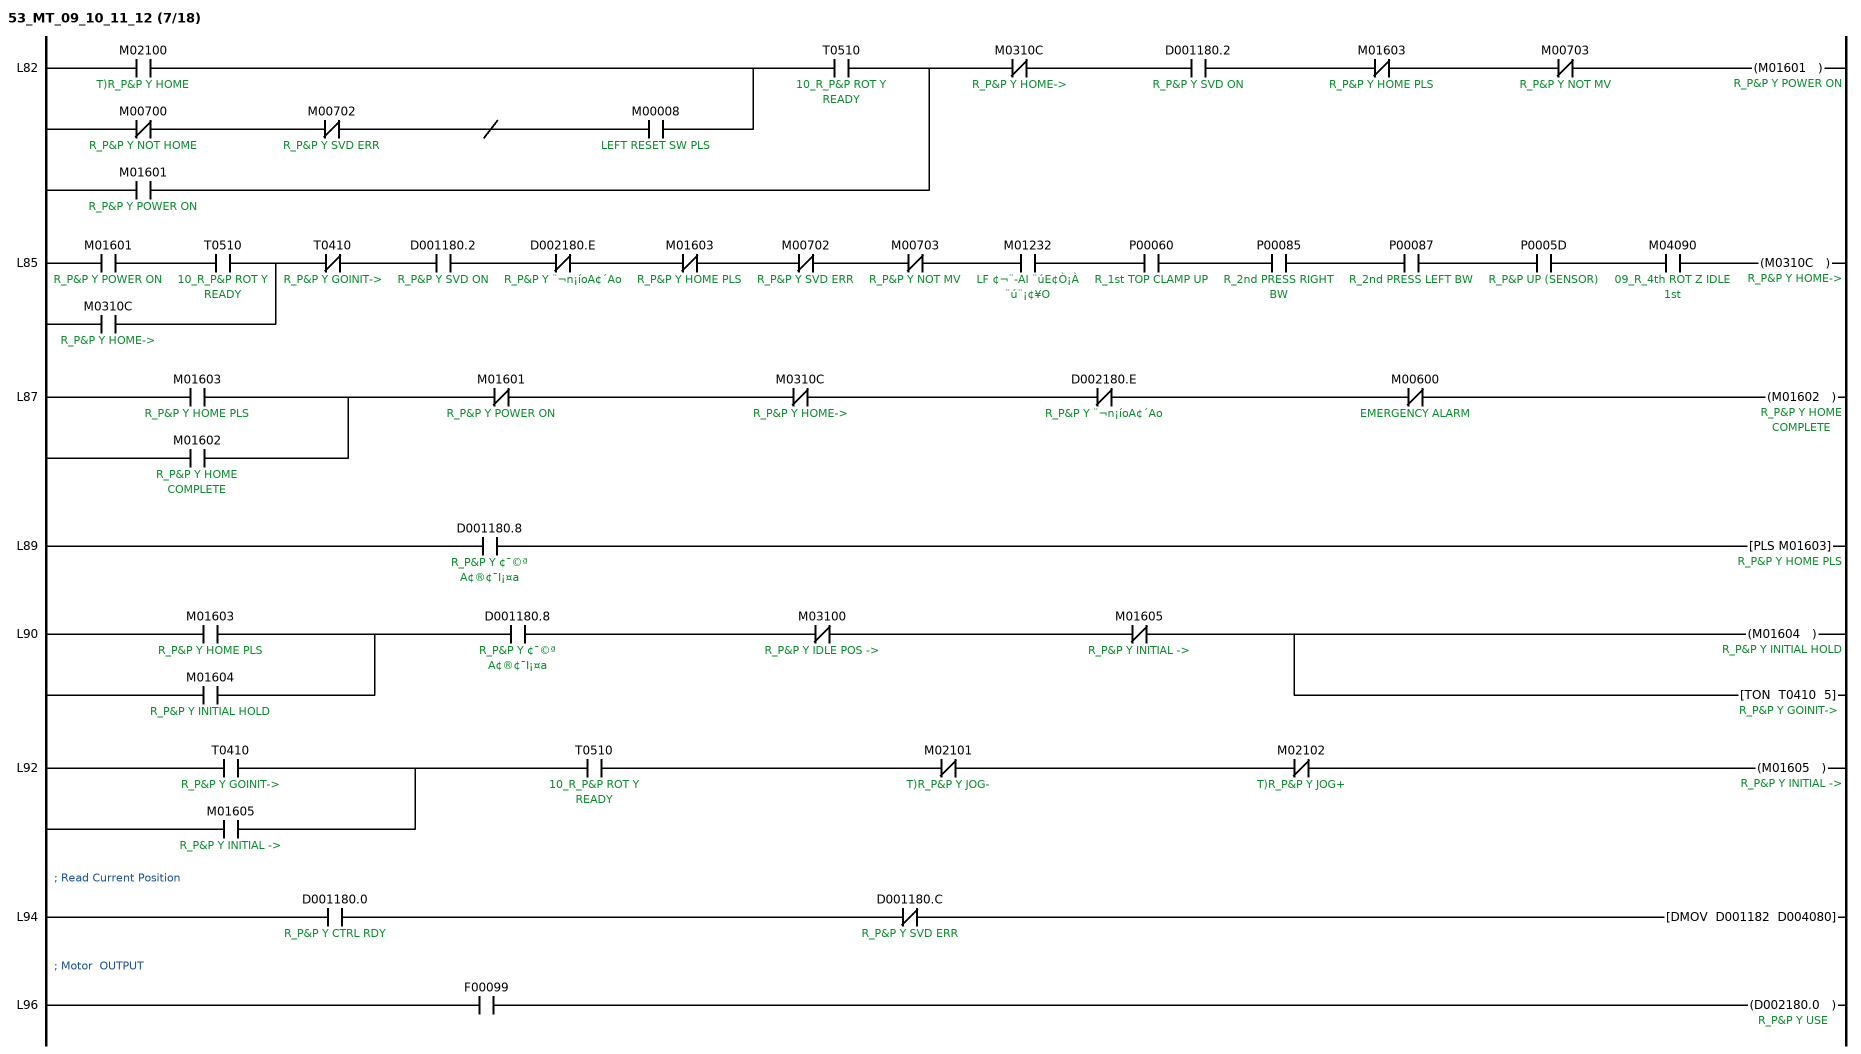
[picture p288: 53_MT_09_10_11_12 rungs L82-L96]
; L82
LOAD      M02100	// T)R_P&P Y HOME
LOAD NOT  M00700	// R_P&P Y NOT HOME
AND NOT   M00702	// R_P&P Y SVD ERR
NOT
AND       M00008	// LEFT RESET SW PLS
OR LOAD
AND       T0510	// 10_R_P&P ROT Y READY
OR        M01601	// R_P&P Y POWER ON
AND NOT   M0310C	// R_P&P Y HOME->
AND       D001180.2	// R_P&P Y SVD ON
AND NOT   M01603	// R_P&P Y HOME PLS
AND NOT   M00703	// R_P&P Y NOT MV
OUT       M01601	// R_P&P Y POWER ON
; L85
LOAD      M01601	// R_P&P Y POWER ON
AND       T0510	// 10_R_P&P ROT Y READY
OR        M0310C	// R_P&P Y HOME->
AND NOT   T0410	// R_P&P Y GOINIT->
AND       D001180.2	// R_P&P Y SVD ON
AND NOT   D002180.E	// R_P&P Y ¨¬n¡íoA¢´Ao
AND NOT   M01603	// R_P&P Y HOME PLS
AND NOT   M00702	// R_P&P Y SVD ERR
AND NOT   M00703	// R_P&P Y NOT MV
AND       M01232	// LF ¢¬¨­AI ¨úE¢Ò¡À ¨ú¨¡¢¥O
AND       P00060	// R_1st TOP CLAMP UP
AND       P00085	// R_2nd PRESS RIGHT BW
AND       P00087	// R_2nd PRESS LEFT BW
AND       P0005D	// R_P&P UP (SENSOR)
AND       M04090	// 09_R_4th ROT Z IDLE 1st
OUT       M0310C	// R_P&P Y HOME->
; L87
LOAD      M01603	// R_P&P Y HOME PLS
OR        M01602	// R_P&P Y HOME COMPLETE
AND NOT   M01601	// R_P&P Y POWER ON
AND NOT   M0310C	// R_P&P Y HOME->
AND NOT   D002180.E	// R_P&P Y ¨¬n¡íoA¢´Ao
AND NOT   M00600	// EMERGENCY ALARM
OUT       M01602	// R_P&P Y HOME COMPLETE
; L89
LOAD      D001180.8	// R_P&P Y ¢¯©ªA¢®¢¯I¡¤a
OUTP      M01603	// R_P&P Y HOME PLS
; L90
LOAD      M01603	// R_P&P Y HOME PLS
OR        M01604	// R_P&P Y INITIAL HOLD
AND       D001180.8	// R_P&P Y ¢¯©ªA¢®¢¯I¡¤a
AND NOT   M03100	// R_P&P Y IDLE POS ->
AND NOT   M01605	// R_P&P Y INITIAL ->
OUT       M01604	// R_P&P Y INITIAL HOLD
TON       T0410 5	// R_P&P Y GOINIT->
; L92
LOAD      T0410	// R_P&P Y GOINIT->
OR        M01605	// R_P&P Y INITIAL ->
AND       T0510	// 10_R_P&P ROT Y READY
AND NOT   M02101	// T)R_P&P Y JOG-
AND NOT   M02102	// T)R_P&P Y JOG+
OUT       M01605	// R_P&P Y INITIAL ->
; L94
LOAD      D001180.0	// R_P&P Y CTRL RDY
AND NOT   D001180.C	// R_P&P Y SVD ERR
DMOV      D001182 D004080
// output comment: Read Current Position
//  Motor  OUTPUT
; L96
LOAD      F00099
OUT       D002180.0	// R_P&P Y USE

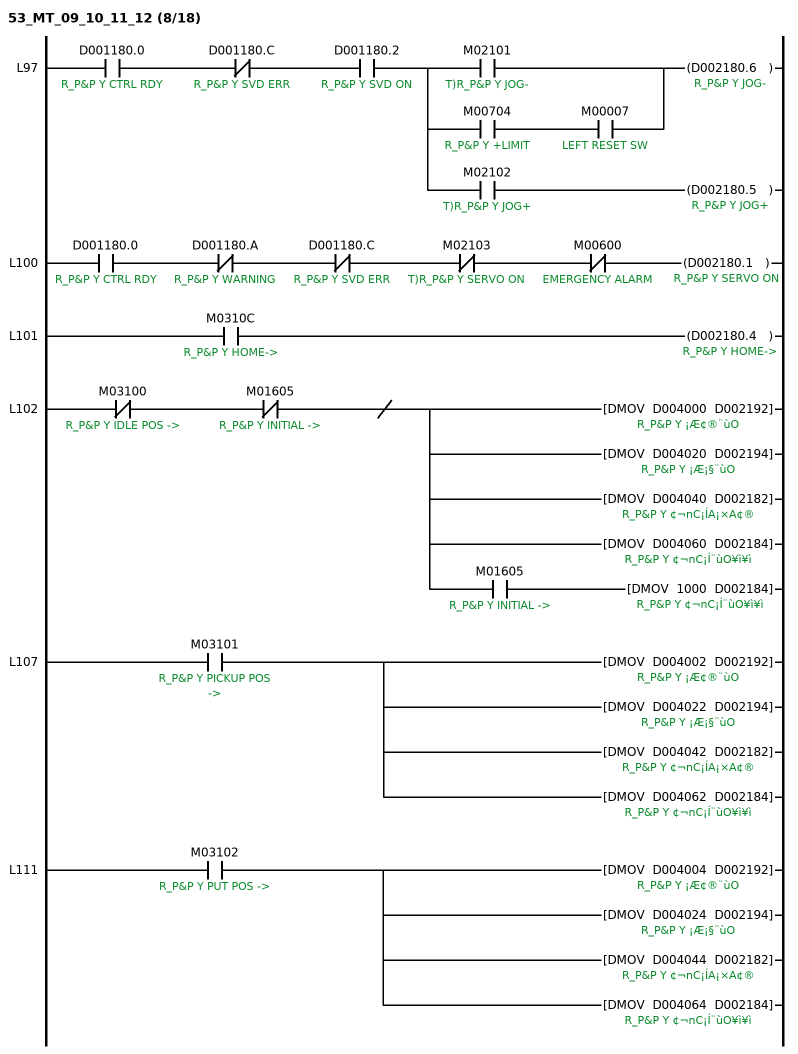
; L97
LOAD      D001180.0	// R_P&P Y CTRL RDY
AND NOT   D001180.C	// R_P&P Y SVD ERR
AND       D001180.2	// R_P&P Y SVD ON
MPUSH
LOAD      M02101	// T)R_P&P Y JOG-
LOAD      M00704	// R_P&P Y +LIMIT
AND       M00007	// LEFT RESET SW
OR LOAD
AND LOAD
OUT       D002180.6	// R_P&P Y JOG-
MPOP
AND       M02102	// T)R_P&P Y JOG+
OUT       D002180.5	// R_P&P Y JOG+
; L100
LOAD      D001180.0	// R_P&P Y CTRL RDY
AND NOT   D001180.A	// R_P&P Y WARNING
AND NOT   D001180.C	// R_P&P Y SVD ERR
AND NOT   M02103	// T)R_P&P Y SERVO ON
AND NOT   M00600	// EMERGENCY ALARM
OUT       D002180.1	// R_P&P Y SERVO ON
; L101
LOAD      M0310C	// R_P&P Y HOME->
OUT       D002180.4	// R_P&P Y HOME->
; L102
LOAD NOT  M03100	// R_P&P Y IDLE POS ->
AND NOT   M01605	// R_P&P Y INITIAL ->
NOT
DMOV      D004000 D002192	// R_P&P Y ¡Æ¢®¨ùO
DMOV      D004020 D002194	// R_P&P Y ¡Æ¡§¨ùO
DMOV      D004040 D002182	// R_P&P Y ¢¬nC¡ÍA¡×A¢®
DMOV      D004060 D002184	// R_P&P Y ¢¬nC¡Í¨ùO¥ì¥ì
AND       M01605	// R_P&P Y INITIAL ->
DMOV      1000 D002184	// R_P&P Y ¢¬nC¡Í¨ùO¥ì¥ì
; L107
LOAD      M03101	// R_P&P Y PICKUP POS ->
DMOV      D004002 D002192	// R_P&P Y ¡Æ¢®¨ùO
DMOV      D004022 D002194	// R_P&P Y ¡Æ¡§¨ùO
DMOV      D004042 D002182	// R_P&P Y ¢¬nC¡ÍA¡×A¢®
DMOV      D004062 D002184	// R_P&P Y ¢¬nC¡Í¨ùO¥ì¥ì
; L111
LOAD      M03102	// R_P&P Y PUT POS ->
DMOV      D004004 D002192	// R_P&P Y ¡Æ¢®¨ùO
DMOV      D004024 D002194	// R_P&P Y ¡Æ¡§¨ùO
DMOV      D004044 D002182	// R_P&P Y ¢¬nC¡ÍA¡×A¢®
DMOV      D004064 D002184	// R_P&P Y ¢¬nC¡Í¨ùO¥ì¥ì

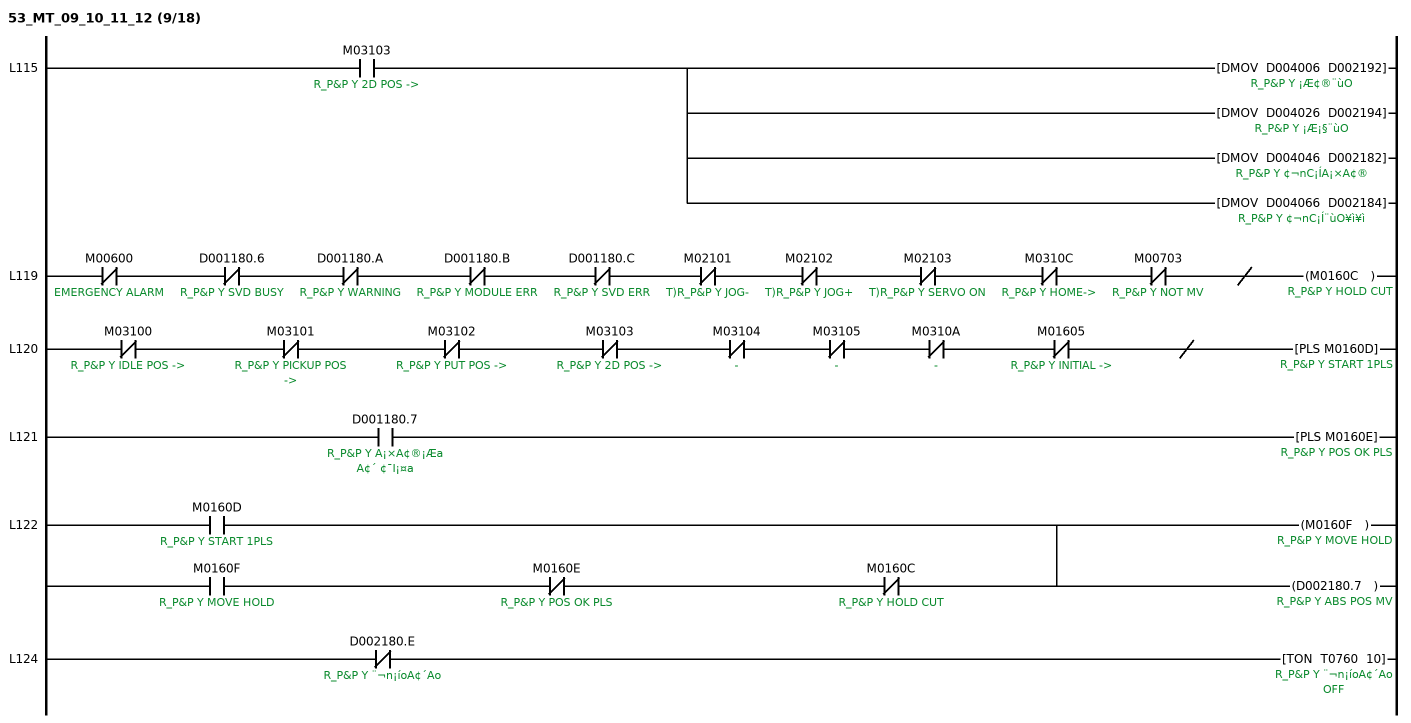
; L115
LOAD      M03103	// R_P&P Y 2D POS ->
DMOV      D004006 D002192	// R_P&P Y ¡Æ¢®¨ùO
DMOV      D004026 D002194	// R_P&P Y ¡Æ¡§¨ùO
DMOV      D004046 D002182	// R_P&P Y ¢¬nC¡ÍA¡×A¢®
DMOV      D004066 D002184	// R_P&P Y ¢¬nC¡Í¨ùO¥ì¥ì
; L119
LOAD NOT  M00600	// EMERGENCY ALARM
AND NOT   D001180.6	// R_P&P Y SVD BUSY
AND NOT   D001180.A	// R_P&P Y WARNING
AND NOT   D001180.B	// R_P&P Y MODULE ERR
AND NOT   D001180.C	// R_P&P Y SVD ERR
AND NOT   M02101	// T)R_P&P Y JOG-
AND NOT   M02102	// T)R_P&P Y JOG+
AND NOT   M02103	// T)R_P&P Y SERVO ON
AND NOT   M0310C	// R_P&P Y HOME->
AND NOT   M00703	// R_P&P Y NOT MV
NOT
OUT       M0160C	// R_P&P Y HOLD CUT
; L120
LOAD NOT  M03100	// R_P&P Y IDLE POS ->
AND NOT   M03101	// R_P&P Y PICKUP POS ->
AND NOT   M03102	// R_P&P Y PUT POS ->
AND NOT   M03103	// R_P&P Y 2D POS ->
AND NOT   M03104	// -
AND NOT   M03105	// -
AND NOT   M0310A	// -
AND NOT   M01605	// R_P&P Y INITIAL ->
NOT
OUTP      M0160D	// R_P&P Y START 1PLS
; L121
LOAD      D001180.7	// R_P&P Y A¡×A¢®¡ÆaA¢´ ¢¯I¡¤a
OUTP      M0160E	// R_P&P Y POS OK PLS
; L122
LOAD      M0160D	// R_P&P Y START 1PLS
LOAD      M0160F	// R_P&P Y MOVE HOLD
AND NOT   M0160E	// R_P&P Y POS OK PLS
AND NOT   M0160C	// R_P&P Y HOLD CUT
OR LOAD
OUT       M0160F	// R_P&P Y MOVE HOLD
OUT       D002180.7	// R_P&P Y ABS POS MV
; L124
LOAD NOT  D002180.E	// R_P&P Y ¨¬n¡íoA¢´Ao
TON       T0760 10	// R_P&P Y ¨¬n¡íoA¢´AoOFF

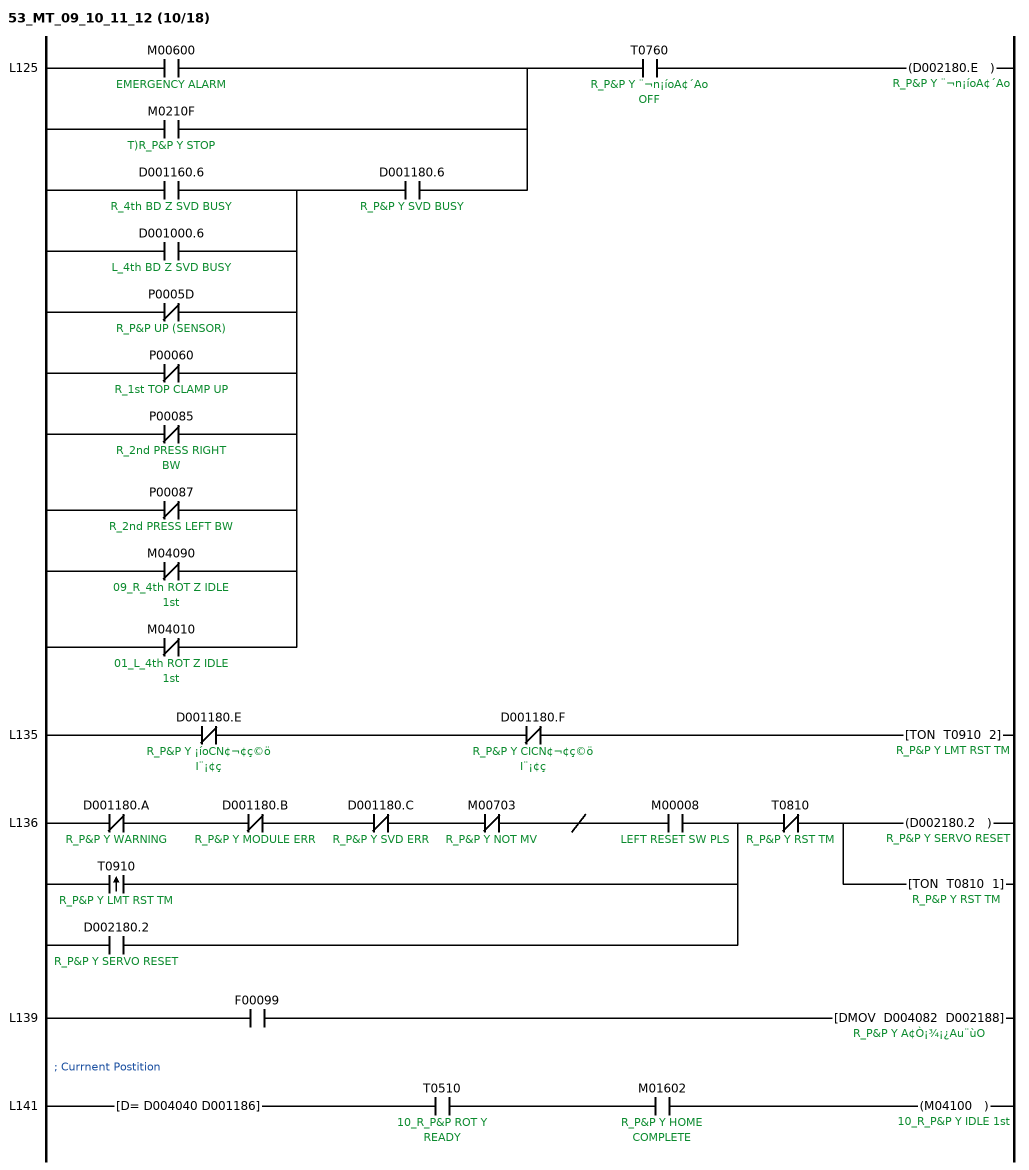
; L125
LOAD      M00600	// EMERGENCY ALARM
OR        M0210F	// T)R_P&P Y STOP
LOAD      D001160.6	// R_4th BD Z SVD BUSY
OR        D001000.6	// L_4th BD Z SVD BUSY
OR NOT    P0005D	// R_P&P UP (SENSOR)
OR NOT    P00060	// R_1st TOP CLAMP UP
OR NOT    P00085	// R_2nd PRESS RIGHT BW
OR NOT    P00087	// R_2nd PRESS LEFT BW
OR NOT    M04090	// 09_R_4th ROT Z IDLE 1st
OR NOT    M04010	// 01_L_4th ROT Z IDLE 1st
AND       D001180.6	// R_P&P Y SVD BUSY
OR LOAD
AND       T0760	// R_P&P Y ¨¬n¡íoA¢´AoOFF
OUT       D002180.E	// R_P&P Y ¨¬n¡íoA¢´Ao
; L135
LOAD NOT  D001180.E	// R_P&P Y ¡íoCN¢¬¢ç©öI¨¡¢ç
AND NOT   D001180.F	// R_P&P Y CICN¢¬¢ç©öI¨¡¢ç
TON       T0910 2	// R_P&P Y LMT RST TM
; L136
LOAD NOT  D001180.A	// R_P&P Y WARNING
AND NOT   D001180.B	// R_P&P Y MODULE ERR
AND NOT   D001180.C	// R_P&P Y SVD ERR
AND NOT   M00703	// R_P&P Y NOT MV
NOT
AND       M00008	// LEFT RESET SW PLS
ORP       T0910	// R_P&P Y LMT RST TM
OR        D002180.2	// R_P&P Y SERVO RESET
AND NOT   T0810	// R_P&P Y RST TM
OUT       D002180.2	// R_P&P Y SERVO RESET
TON       T0810 1	// R_P&P Y RST TM
; L139
LOAD      F00099
DMOV      D004082 D002188	// R_P&P Y A¢Ò¡¾¡¿Au¨ùO
// Currnent Postition
; L141
LOADD=    D004040 D001186
AND       T0510	// 10_R_P&P ROT Y READY
AND       M01602	// R_P&P Y HOME COMPLETE
OUT       M04100	// 10_R_P&P Y IDLE 1st

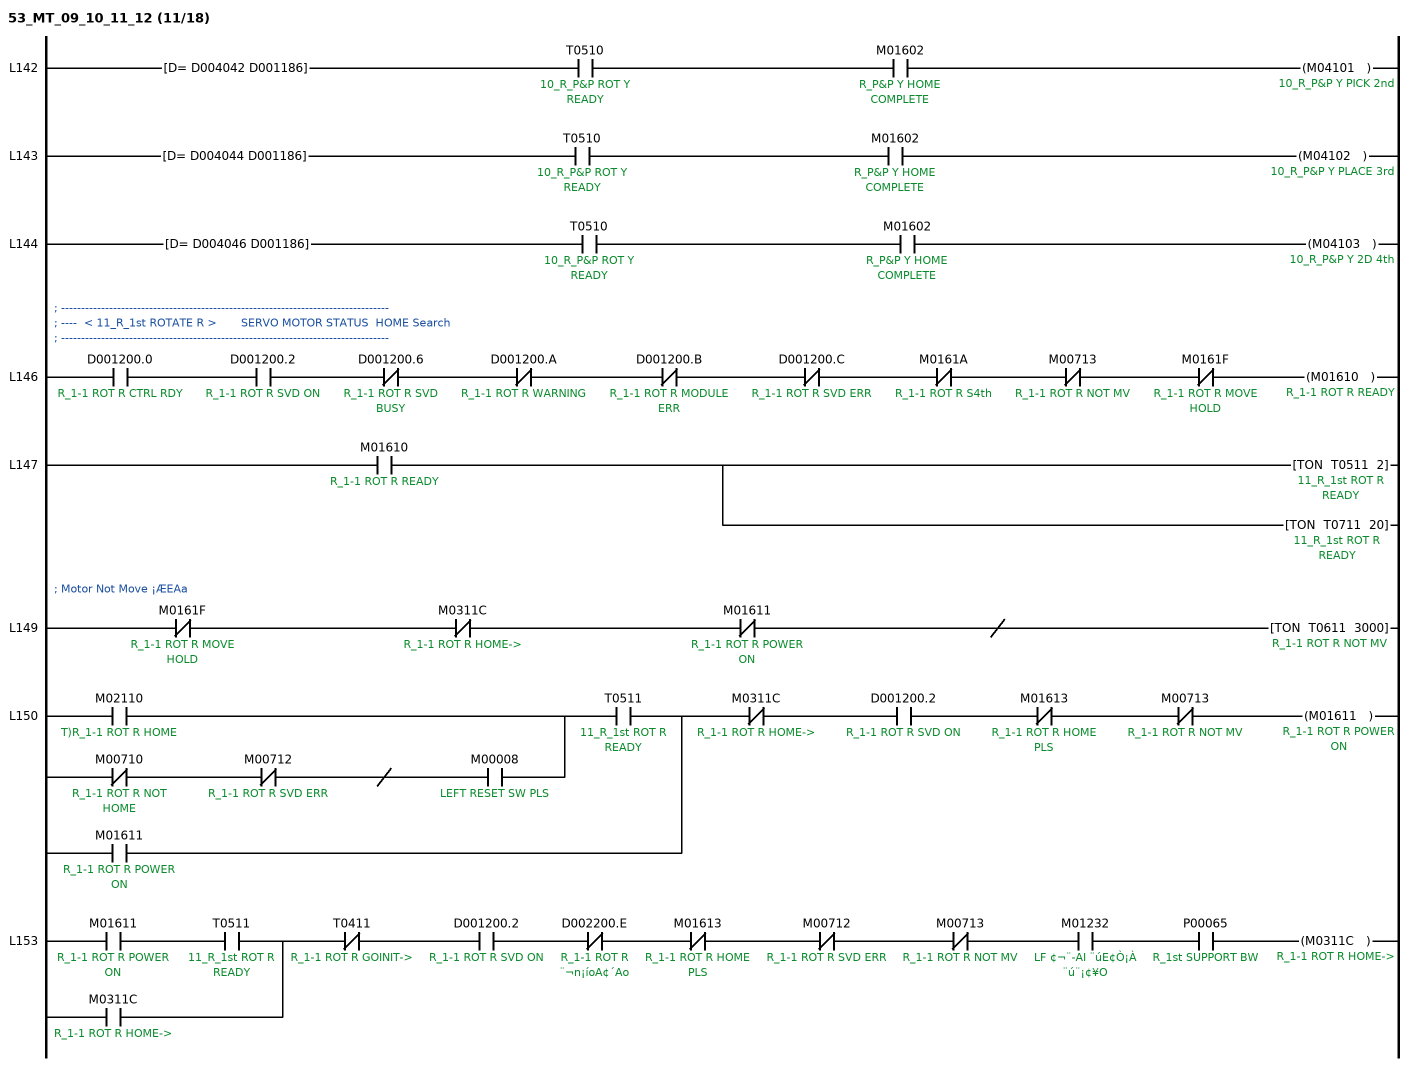
; L142
LOADD=    D004042 D001186
AND       T0510	// 10_R_P&P ROT Y READY
AND       M01602	// R_P&P Y HOME COMPLETE
OUT       M04101	// 10_R_P&P Y PICK 2nd
; L143
LOADD=    D004044 D001186
AND       T0510	// 10_R_P&P ROT Y READY
AND       M01602	// R_P&P Y HOME COMPLETE
OUT       M04102	// 10_R_P&P Y PLACE 3rd
; L144
LOADD=    D004046 D001186
AND       T0510	// 10_R_P&P ROT Y READY
AND       M01602	// R_P&P Y HOME COMPLETE
OUT       M04103	// 10_R_P&P Y 2D 4th
// ----------------------------------------------------------------------------------
// 
// ----  < 11_R_1st ROTATE R >       SERVO MOTOR STATUS  HOME Search
// 
// ----------------------------------------------------------------------------------
; L146
LOAD      D001200.0	// R_1-1 ROT R CTRL RDY
AND       D001200.2	// R_1-1 ROT R SVD ON
AND NOT   D001200.6	// R_1-1 ROT R SVD BUSY
AND NOT   D001200.A	// R_1-1 ROT R WARNING
AND NOT   D001200.B	// R_1-1 ROT R MODULE ERR
AND NOT   D001200.C	// R_1-1 ROT R SVD ERR
AND NOT   M0161A	// R_1-1 ROT R S4th
AND NOT   M00713	// R_1-1 ROT R NOT MV
AND NOT   M0161F	// R_1-1 ROT R MOVE HOLD
OUT       M01610	// R_1-1 ROT R READY
; L147
LOAD      M01610	// R_1-1 ROT R READY
TON       T0511 2	// 11_R_1st ROT R READY
TON       T0711 20	// 11_R_1st ROT R READY
; L149
LOAD NOT  M0161F	// R_1-1 ROT R MOVE HOLD
AND NOT   M0311C	// R_1-1 ROT R HOME->
AND NOT   M01611	// R_1-1 ROT R POWER ON
NOT
TON       T0611 3000	// R_1-1 ROT R NOT MV
// output comment: Motor Not Move ¡ÆEAa
; L150
LOAD      M02110	// T)R_1-1 ROT R HOME
LOAD NOT  M00710	// R_1-1 ROT R NOT HOME
AND NOT   M00712	// R_1-1 ROT R SVD ERR
NOT
AND       M00008	// LEFT RESET SW PLS
OR LOAD
AND       T0511	// 11_R_1st ROT R READY
OR        M01611	// R_1-1 ROT R POWER ON
AND NOT   M0311C	// R_1-1 ROT R HOME->
AND       D001200.2	// R_1-1 ROT R SVD ON
AND NOT   M01613	// R_1-1 ROT R HOME PLS
AND NOT   M00713	// R_1-1 ROT R NOT MV
OUT       M01611	// R_1-1 ROT R POWER ON
; L153
LOAD      M01611	// R_1-1 ROT R POWER ON
AND       T0511	// 11_R_1st ROT R READY
OR        M0311C	// R_1-1 ROT R HOME->
AND NOT   T0411	// R_1-1 ROT R GOINIT->
AND       D001200.2	// R_1-1 ROT R SVD ON
AND NOT   D002200.E	// R_1-1 ROT R ¨¬n¡íoA¢´Ao
AND NOT   M01613	// R_1-1 ROT R HOME PLS
AND NOT   M00712	// R_1-1 ROT R SVD ERR
AND NOT   M00713	// R_1-1 ROT R NOT MV
AND       M01232	// LF ¢¬¨­AI ¨úE¢Ò¡À ¨ú¨¡¢¥O
AND       P00065	// R_1st SUPPORT BW
OUT       M0311C	// R_1-1 ROT R HOME->

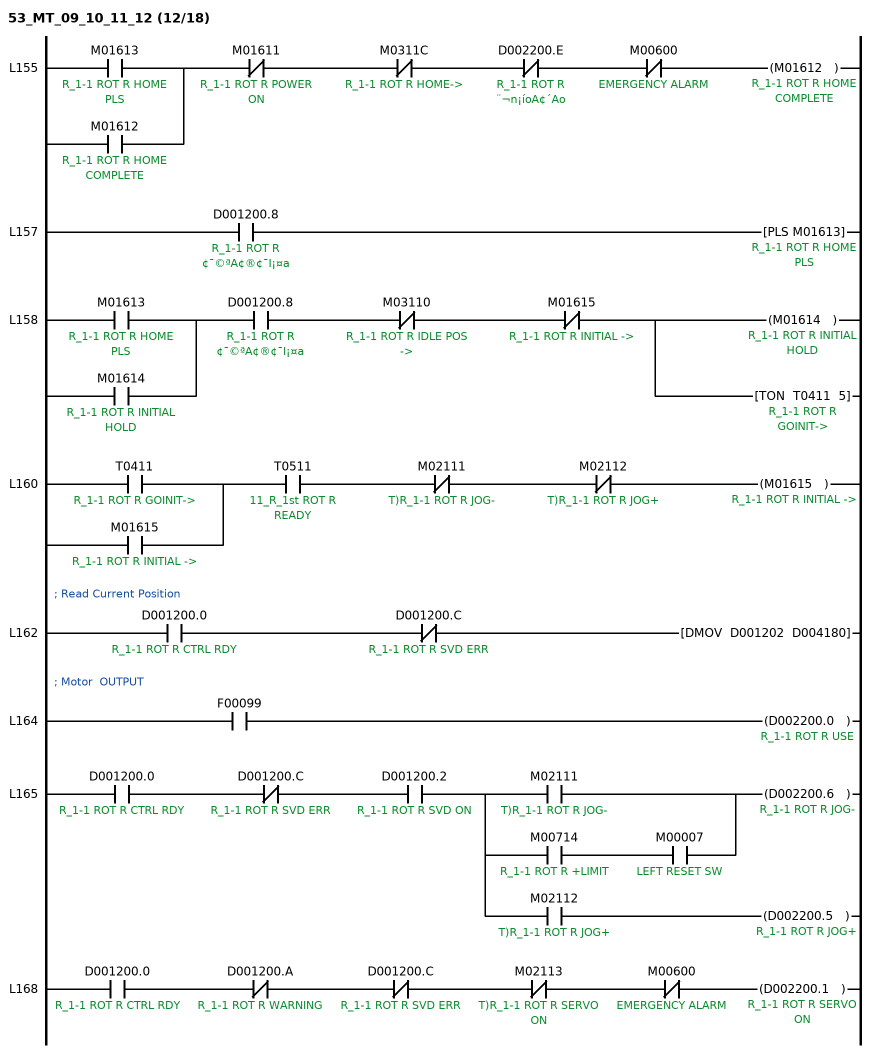
; L155
LOAD      M01613	// R_1-1 ROT R HOME PLS
OR        M01612	// R_1-1 ROT R HOME COMPLETE
AND NOT   M01611	// R_1-1 ROT R POWER ON
AND NOT   M0311C	// R_1-1 ROT R HOME->
AND NOT   D002200.E	// R_1-1 ROT R ¨¬n¡íoA¢´Ao
AND NOT   M00600	// EMERGENCY ALARM
OUT       M01612	// R_1-1 ROT R HOME COMPLETE
; L157
LOAD      D001200.8	// R_1-1 ROT R ¢¯©ªA¢®¢¯I¡¤a
OUTP      M01613	// R_1-1 ROT R HOME PLS
; L158
LOAD      M01613	// R_1-1 ROT R HOME PLS
OR        M01614	// R_1-1 ROT R INITIAL HOLD
AND       D001200.8	// R_1-1 ROT R ¢¯©ªA¢®¢¯I¡¤a
AND NOT   M03110	// R_1-1 ROT R IDLE POS ->
AND NOT   M01615	// R_1-1 ROT R INITIAL ->
OUT       M01614	// R_1-1 ROT R INITIAL HOLD
TON       T0411 5	// R_1-1 ROT R GOINIT->
; L160
LOAD      T0411	// R_1-1 ROT R GOINIT->
OR        M01615	// R_1-1 ROT R INITIAL ->
AND       T0511	// 11_R_1st ROT R READY
AND NOT   M02111	// T)R_1-1 ROT R JOG-
AND NOT   M02112	// T)R_1-1 ROT R JOG+
OUT       M01615	// R_1-1 ROT R INITIAL ->
; L162
LOAD      D001200.0	// R_1-1 ROT R CTRL RDY
AND NOT   D001200.C	// R_1-1 ROT R SVD ERR
DMOV      D001202 D004180
// output comment: Read Current Position
//  Motor  OUTPUT
; L164
LOAD      F00099
OUT       D002200.0	// R_1-1 ROT R USE
; L165
LOAD      D001200.0	// R_1-1 ROT R CTRL RDY
AND NOT   D001200.C	// R_1-1 ROT R SVD ERR
AND       D001200.2	// R_1-1 ROT R SVD ON
MPUSH
LOAD      M02111	// T)R_1-1 ROT R JOG-
LOAD      M00714	// R_1-1 ROT R +LIMIT
AND       M00007	// LEFT RESET SW
OR LOAD
AND LOAD
OUT       D002200.6	// R_1-1 ROT R JOG-
MPOP
AND       M02112	// T)R_1-1 ROT R JOG+
OUT       D002200.5	// R_1-1 ROT R JOG+
; L168
LOAD      D001200.0	// R_1-1 ROT R CTRL RDY
AND NOT   D001200.A	// R_1-1 ROT R WARNING
AND NOT   D001200.C	// R_1-1 ROT R SVD ERR
AND NOT   M02113	// T)R_1-1 ROT R SERVO ON
AND NOT   M00600	// EMERGENCY ALARM
OUT       D002200.1	// R_1-1 ROT R SERVO ON

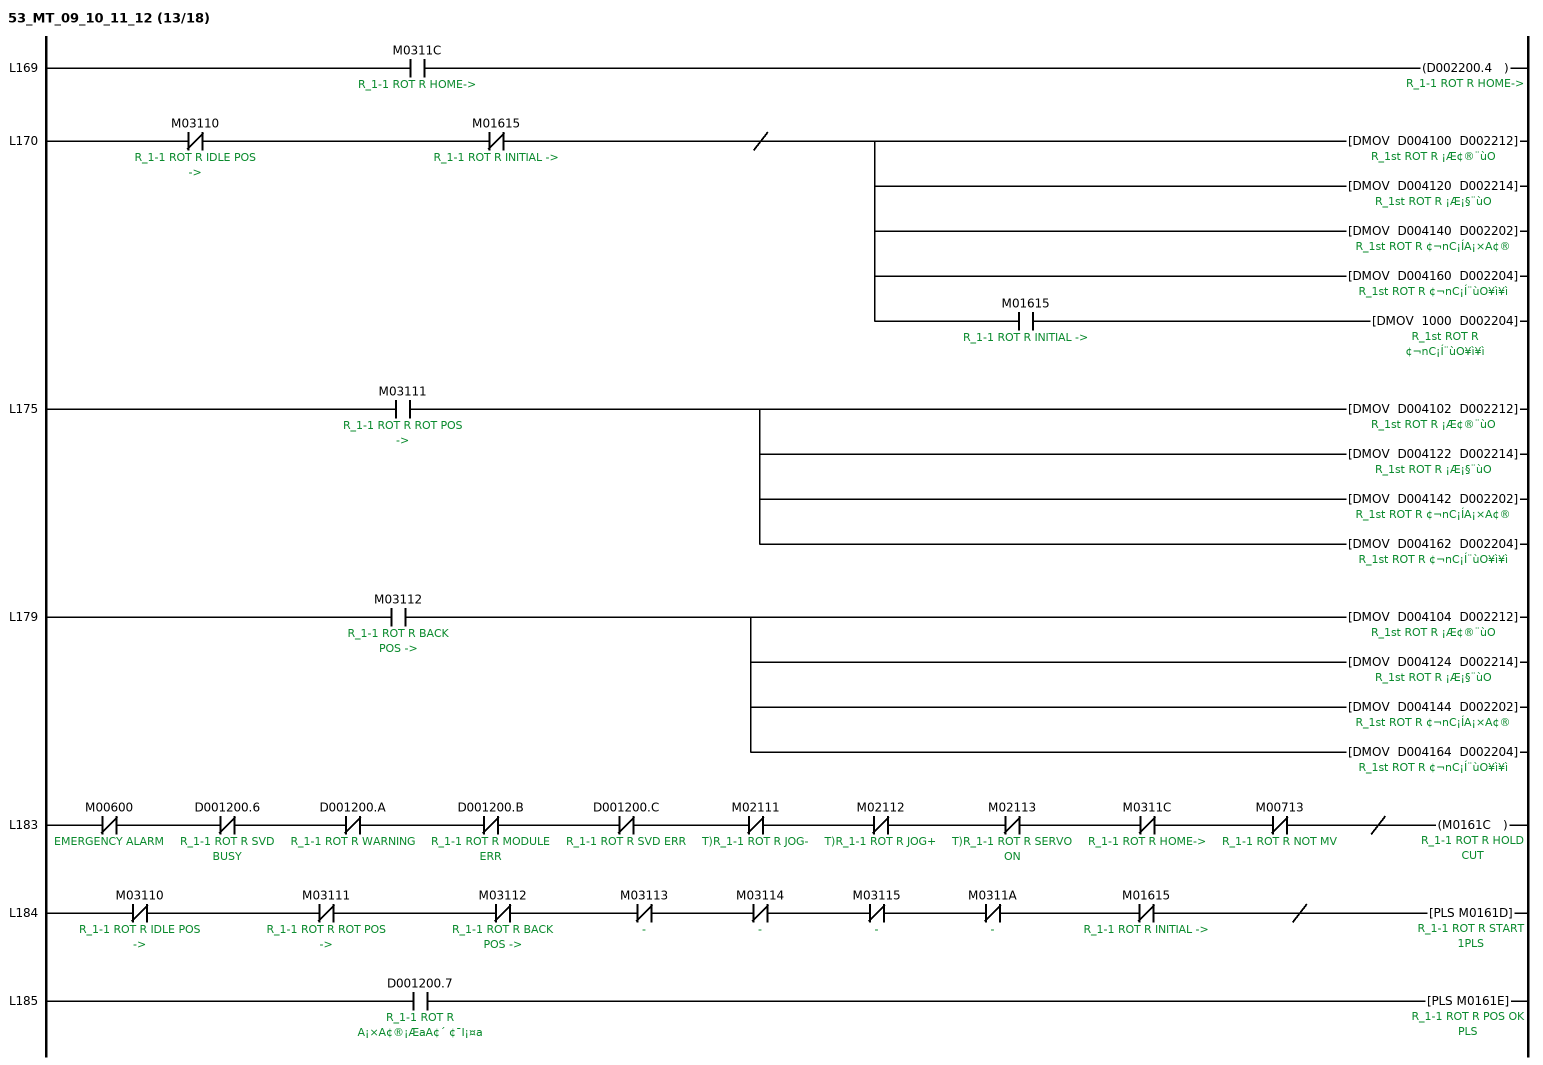
; L169
LOAD      M0311C	// R_1-1 ROT R HOME->
OUT       D002200.4	// R_1-1 ROT R HOME->
; L170
LOAD NOT  M03110	// R_1-1 ROT R IDLE POS ->
AND NOT   M01615	// R_1-1 ROT R INITIAL ->
NOT
DMOV      D004100 D002212	// R_1st ROT R ¡Æ¢®¨ùO
DMOV      D004120 D002214	// R_1st ROT R ¡Æ¡§¨ùO
DMOV      D004140 D002202	// R_1st ROT R ¢¬nC¡ÍA¡×A¢®
DMOV      D004160 D002204	// R_1st ROT R ¢¬nC¡Í¨ùO¥ì¥ì
AND       M01615	// R_1-1 ROT R INITIAL ->
DMOV      1000 D002204	// R_1st ROT R ¢¬nC¡Í¨ùO¥ì¥ì
; L175
LOAD      M03111	// R_1-1 ROT R ROT POS ->
DMOV      D004102 D002212	// R_1st ROT R ¡Æ¢®¨ùO
DMOV      D004122 D002214	// R_1st ROT R ¡Æ¡§¨ùO
DMOV      D004142 D002202	// R_1st ROT R ¢¬nC¡ÍA¡×A¢®
DMOV      D004162 D002204	// R_1st ROT R ¢¬nC¡Í¨ùO¥ì¥ì
; L179
LOAD      M03112	// R_1-1 ROT R BACK POS ->
DMOV      D004104 D002212	// R_1st ROT R ¡Æ¢®¨ùO
DMOV      D004124 D002214	// R_1st ROT R ¡Æ¡§¨ùO
DMOV      D004144 D002202	// R_1st ROT R ¢¬nC¡ÍA¡×A¢®
DMOV      D004164 D002204	// R_1st ROT R ¢¬nC¡Í¨ùO¥ì¥ì
; L183
LOAD NOT  M00600	// EMERGENCY ALARM
AND NOT   D001200.6	// R_1-1 ROT R SVD BUSY
AND NOT   D001200.A	// R_1-1 ROT R WARNING
AND NOT   D001200.B	// R_1-1 ROT R MODULE ERR
AND NOT   D001200.C	// R_1-1 ROT R SVD ERR
AND NOT   M02111	// T)R_1-1 ROT R JOG-
AND NOT   M02112	// T)R_1-1 ROT R JOG+
AND NOT   M02113	// T)R_1-1 ROT R SERVO ON
AND NOT   M0311C	// R_1-1 ROT R HOME->
AND NOT   M00713	// R_1-1 ROT R NOT MV
NOT
OUT       M0161C	// R_1-1 ROT R HOLD CUT
; L184
LOAD NOT  M03110	// R_1-1 ROT R IDLE POS ->
AND NOT   M03111	// R_1-1 ROT R ROT POS ->
AND NOT   M03112	// R_1-1 ROT R BACK POS ->
AND NOT   M03113	// -
AND NOT   M03114	// -
AND NOT   M03115	// -
AND NOT   M0311A	// -
AND NOT   M01615	// R_1-1 ROT R INITIAL ->
NOT
OUTP      M0161D	// R_1-1 ROT R START 1PLS
; L185
LOAD      D001200.7	// R_1-1 ROT R A¡×A¢®¡ÆaA¢´ ¢¯I¡¤a
OUTP      M0161E	// R_1-1 ROT R POS OK PLS

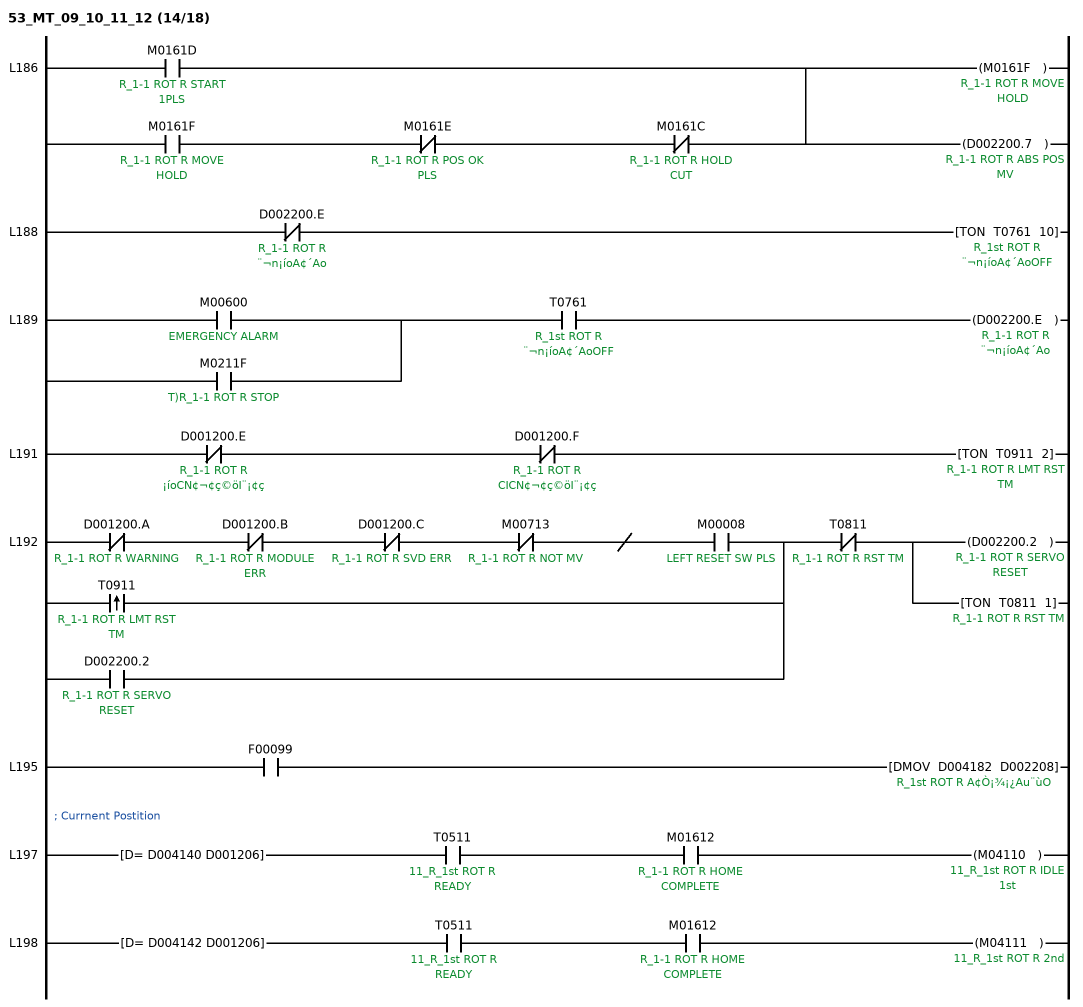
; L186
LOAD      M0161D	// R_1-1 ROT R START 1PLS
LOAD      M0161F	// R_1-1 ROT R MOVE HOLD
AND NOT   M0161E	// R_1-1 ROT R POS OK PLS
AND NOT   M0161C	// R_1-1 ROT R HOLD CUT
OR LOAD
OUT       M0161F	// R_1-1 ROT R MOVE HOLD
OUT       D002200.7	// R_1-1 ROT R ABS POS MV
; L188
LOAD NOT  D002200.E	// R_1-1 ROT R ¨¬n¡íoA¢´Ao
TON       T0761 10	// R_1st ROT R ¨¬n¡íoA¢´AoOFF
; L189
LOAD      M00600	// EMERGENCY ALARM
OR        M0211F	// T)R_1-1 ROT R STOP
AND       T0761	// R_1st ROT R ¨¬n¡íoA¢´AoOFF
OUT       D002200.E	// R_1-1 ROT R ¨¬n¡íoA¢´Ao
; L191
LOAD NOT  D001200.E	// R_1-1 ROT R ¡íoCN¢¬¢ç©öI¨¡¢ç
AND NOT   D001200.F	// R_1-1 ROT R CICN¢¬¢ç©öI¨¡¢ç
TON       T0911 2	// R_1-1 ROT R LMT RST TM
; L192
LOAD NOT  D001200.A	// R_1-1 ROT R WARNING
AND NOT   D001200.B	// R_1-1 ROT R MODULE ERR
AND NOT   D001200.C	// R_1-1 ROT R SVD ERR
AND NOT   M00713	// R_1-1 ROT R NOT MV
NOT
AND       M00008	// LEFT RESET SW PLS
ORP       T0911	// R_1-1 ROT R LMT RST TM
OR        D002200.2	// R_1-1 ROT R SERVO RESET
AND NOT   T0811	// R_1-1 ROT R RST TM
OUT       D002200.2	// R_1-1 ROT R SERVO RESET
TON       T0811 1	// R_1-1 ROT R RST TM
; L195
LOAD      F00099
DMOV      D004182 D002208	// R_1st ROT R A¢Ò¡¾¡¿Au¨ùO
// Currnent Postition
; L197
LOADD=    D004140 D001206
AND       T0511	// 11_R_1st ROT R READY
AND       M01612	// R_1-1 ROT R HOME COMPLETE
OUT       M04110	// 11_R_1st ROT R IDLE 1st
; L198
LOADD=    D004142 D001206
AND       T0511	// 11_R_1st ROT R READY
AND       M01612	// R_1-1 ROT R HOME COMPLETE
OUT       M04111	// 11_R_1st ROT R 2nd

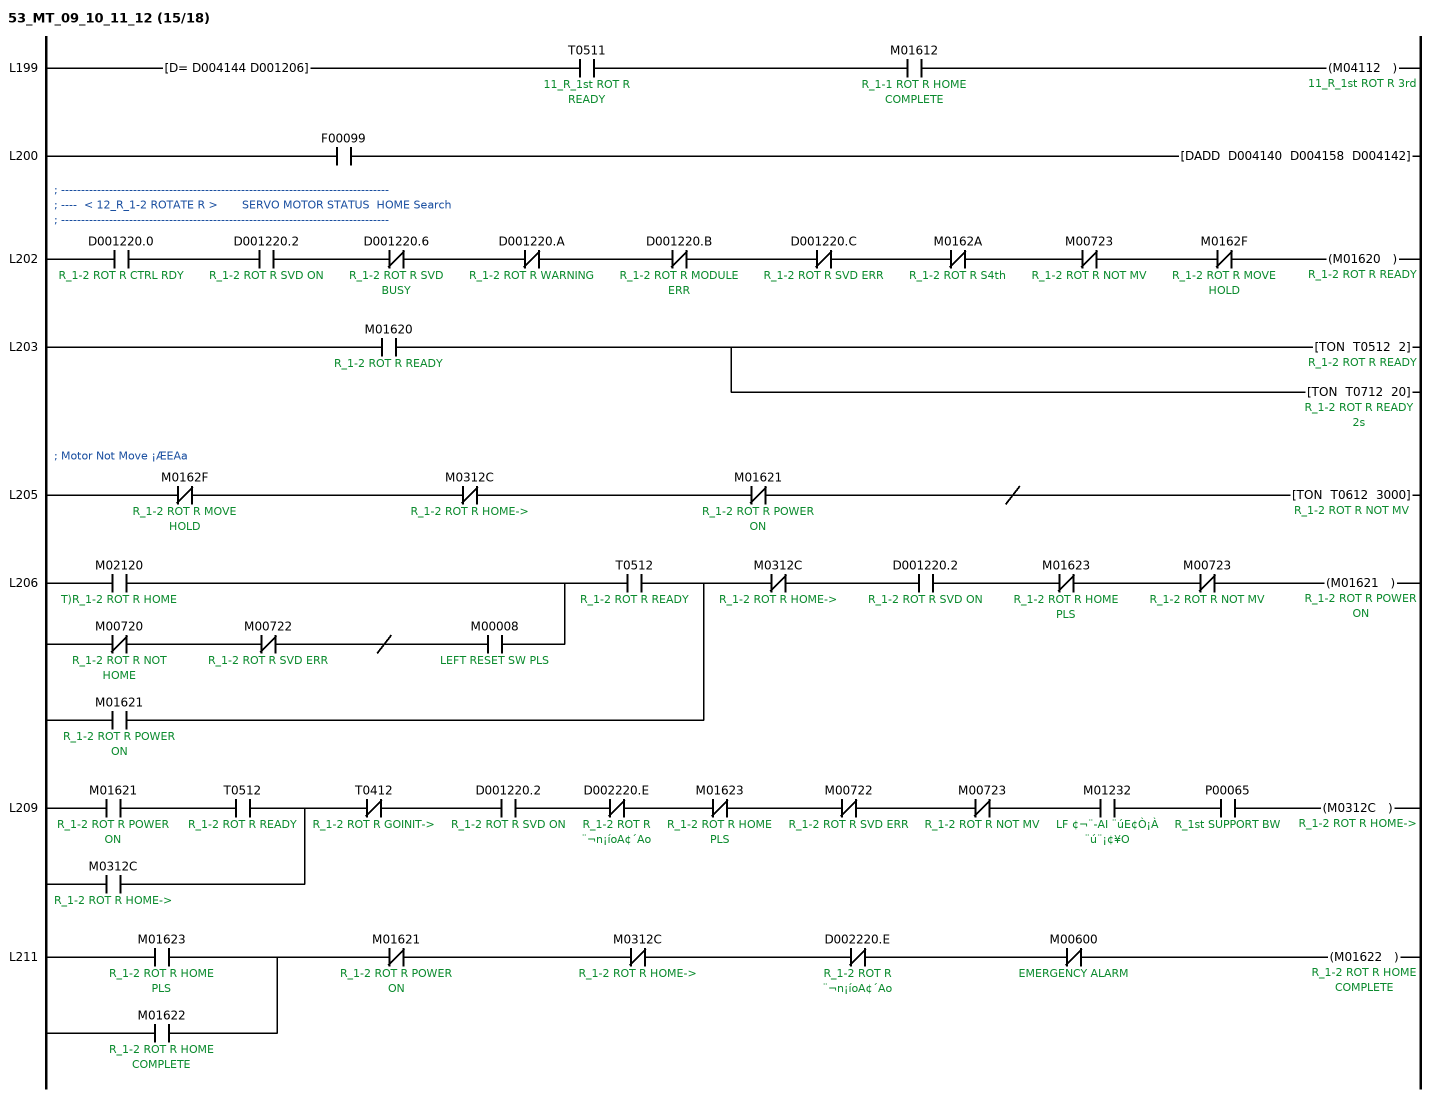
; L199
LOADD=    D004144 D001206
AND       T0511	// 11_R_1st ROT R READY
AND       M01612	// R_1-1 ROT R HOME COMPLETE
OUT       M04112	// 11_R_1st ROT R 3rd
; L200
LOAD      F00099
DADD      D004140 D004158 D004142
// ----------------------------------------------------------------------------------
// 
// ----  < 12_R_1-2 ROTATE R >       SERVO MOTOR STATUS  HOME Search
// 
// ----------------------------------------------------------------------------------
; L202
LOAD      D001220.0	// R_1-2 ROT R CTRL RDY
AND       D001220.2	// R_1-2 ROT R SVD ON
AND NOT   D001220.6	// R_1-2 ROT R SVD BUSY
AND NOT   D001220.A	// R_1-2 ROT R WARNING
AND NOT   D001220.B	// R_1-2 ROT R MODULE ERR
AND NOT   D001220.C	// R_1-2 ROT R SVD ERR
AND NOT   M0162A	// R_1-2 ROT R S4th
AND NOT   M00723	// R_1-2 ROT R NOT MV
AND NOT   M0162F	// R_1-2 ROT R MOVE HOLD
OUT       M01620	// R_1-2 ROT R READY
; L203
LOAD      M01620	// R_1-2 ROT R READY
TON       T0512 2	// R_1-2 ROT R READY
TON       T0712 20	// R_1-2 ROT R READY 2s
; L205
LOAD NOT  M0162F	// R_1-2 ROT R MOVE HOLD
AND NOT   M0312C	// R_1-2 ROT R HOME->
AND NOT   M01621	// R_1-2 ROT R POWER ON
NOT
TON       T0612 3000	// R_1-2 ROT R NOT MV
// output comment: Motor Not Move ¡ÆEAa
; L206
LOAD      M02120	// T)R_1-2 ROT R HOME
LOAD NOT  M00720	// R_1-2 ROT R NOT HOME
AND NOT   M00722	// R_1-2 ROT R SVD ERR
NOT
AND       M00008	// LEFT RESET SW PLS
OR LOAD
AND       T0512	// R_1-2 ROT R READY
OR        M01621	// R_1-2 ROT R POWER ON
AND NOT   M0312C	// R_1-2 ROT R HOME->
AND       D001220.2	// R_1-2 ROT R SVD ON
AND NOT   M01623	// R_1-2 ROT R HOME PLS
AND NOT   M00723	// R_1-2 ROT R NOT MV
OUT       M01621	// R_1-2 ROT R POWER ON
; L209
LOAD      M01621	// R_1-2 ROT R POWER ON
AND       T0512	// R_1-2 ROT R READY
OR        M0312C	// R_1-2 ROT R HOME->
AND NOT   T0412	// R_1-2 ROT R GOINIT->
AND       D001220.2	// R_1-2 ROT R SVD ON
AND NOT   D002220.E	// R_1-2 ROT R ¨¬n¡íoA¢´Ao
AND NOT   M01623	// R_1-2 ROT R HOME PLS
AND NOT   M00722	// R_1-2 ROT R SVD ERR
AND NOT   M00723	// R_1-2 ROT R NOT MV
AND       M01232	// LF ¢¬¨­AI ¨úE¢Ò¡À ¨ú¨¡¢¥O
AND       P00065	// R_1st SUPPORT BW
OUT       M0312C	// R_1-2 ROT R HOME->
; L211
LOAD      M01623	// R_1-2 ROT R HOME PLS
OR        M01622	// R_1-2 ROT R HOME COMPLETE
AND NOT   M01621	// R_1-2 ROT R POWER ON
AND NOT   M0312C	// R_1-2 ROT R HOME->
AND NOT   D002220.E	// R_1-2 ROT R ¨¬n¡íoA¢´Ao
AND NOT   M00600	// EMERGENCY ALARM
OUT       M01622	// R_1-2 ROT R HOME COMPLETE

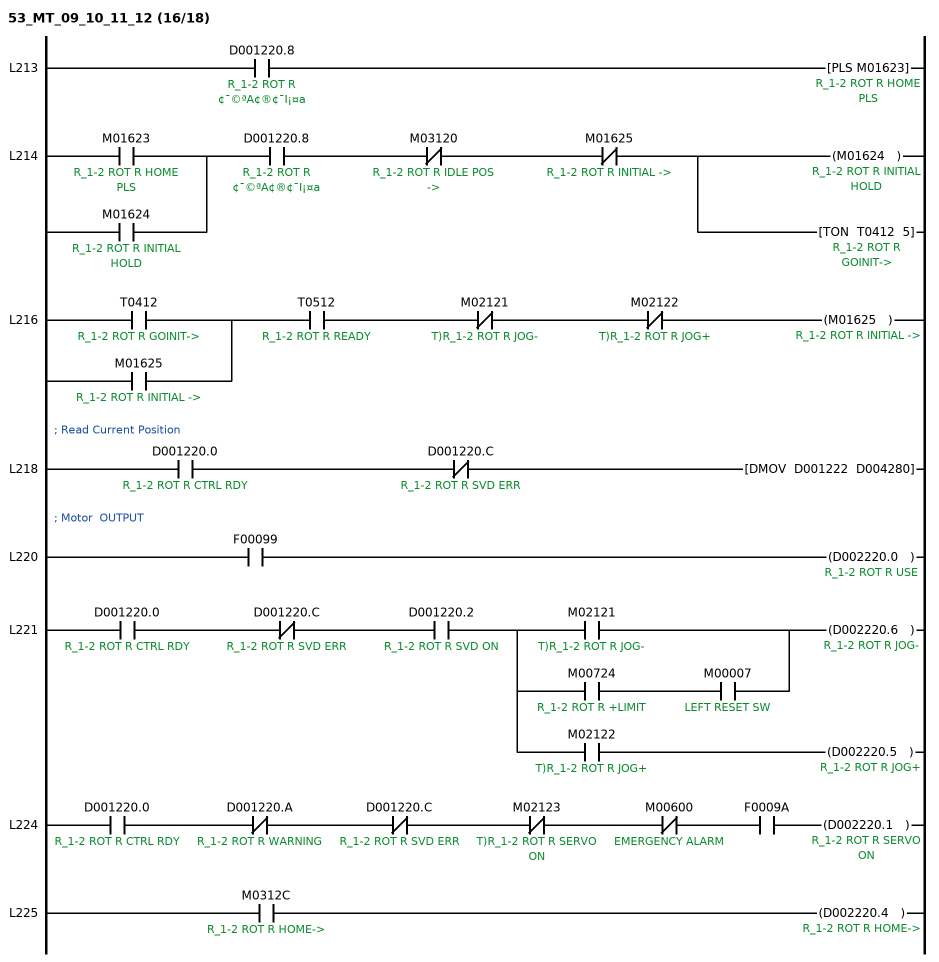
; L213
LOAD      D001220.8	// R_1-2 ROT R ¢¯©ªA¢®¢¯I¡¤a
OUTP      M01623	// R_1-2 ROT R HOME PLS
; L214
LOAD      M01623	// R_1-2 ROT R HOME PLS
OR        M01624	// R_1-2 ROT R INITIAL HOLD
AND       D001220.8	// R_1-2 ROT R ¢¯©ªA¢®¢¯I¡¤a
AND NOT   M03120	// R_1-2 ROT R IDLE POS ->
AND NOT   M01625	// R_1-2 ROT R INITIAL ->
OUT       M01624	// R_1-2 ROT R INITIAL HOLD
TON       T0412 5	// R_1-2 ROT R GOINIT->
; L216
LOAD      T0412	// R_1-2 ROT R GOINIT->
OR        M01625	// R_1-2 ROT R INITIAL ->
AND       T0512	// R_1-2 ROT R READY
AND NOT   M02121	// T)R_1-2 ROT R JOG-
AND NOT   M02122	// T)R_1-2 ROT R JOG+
OUT       M01625	// R_1-2 ROT R INITIAL ->
; L218
LOAD      D001220.0	// R_1-2 ROT R CTRL RDY
AND NOT   D001220.C	// R_1-2 ROT R SVD ERR
DMOV      D001222 D004280
// output comment: Read Current Position
//  Motor  OUTPUT
; L220
LOAD      F00099
OUT       D002220.0	// R_1-2 ROT R USE
; L221
LOAD      D001220.0	// R_1-2 ROT R CTRL RDY
AND NOT   D001220.C	// R_1-2 ROT R SVD ERR
AND       D001220.2	// R_1-2 ROT R SVD ON
MPUSH
LOAD      M02121	// T)R_1-2 ROT R JOG-
LOAD      M00724	// R_1-2 ROT R +LIMIT
AND       M00007	// LEFT RESET SW
OR LOAD
AND LOAD
OUT       D002220.6	// R_1-2 ROT R JOG-
MPOP
AND       M02122	// T)R_1-2 ROT R JOG+
OUT       D002220.5	// R_1-2 ROT R JOG+
; L224
LOAD      D001220.0	// R_1-2 ROT R CTRL RDY
AND NOT   D001220.A	// R_1-2 ROT R WARNING
AND NOT   D001220.C	// R_1-2 ROT R SVD ERR
AND NOT   M02123	// T)R_1-2 ROT R SERVO ON
AND NOT   M00600	// EMERGENCY ALARM
AND       F0009A
OUT       D002220.1	// R_1-2 ROT R SERVO ON
; L225
LOAD      M0312C	// R_1-2 ROT R HOME->
OUT       D002220.4	// R_1-2 ROT R HOME->

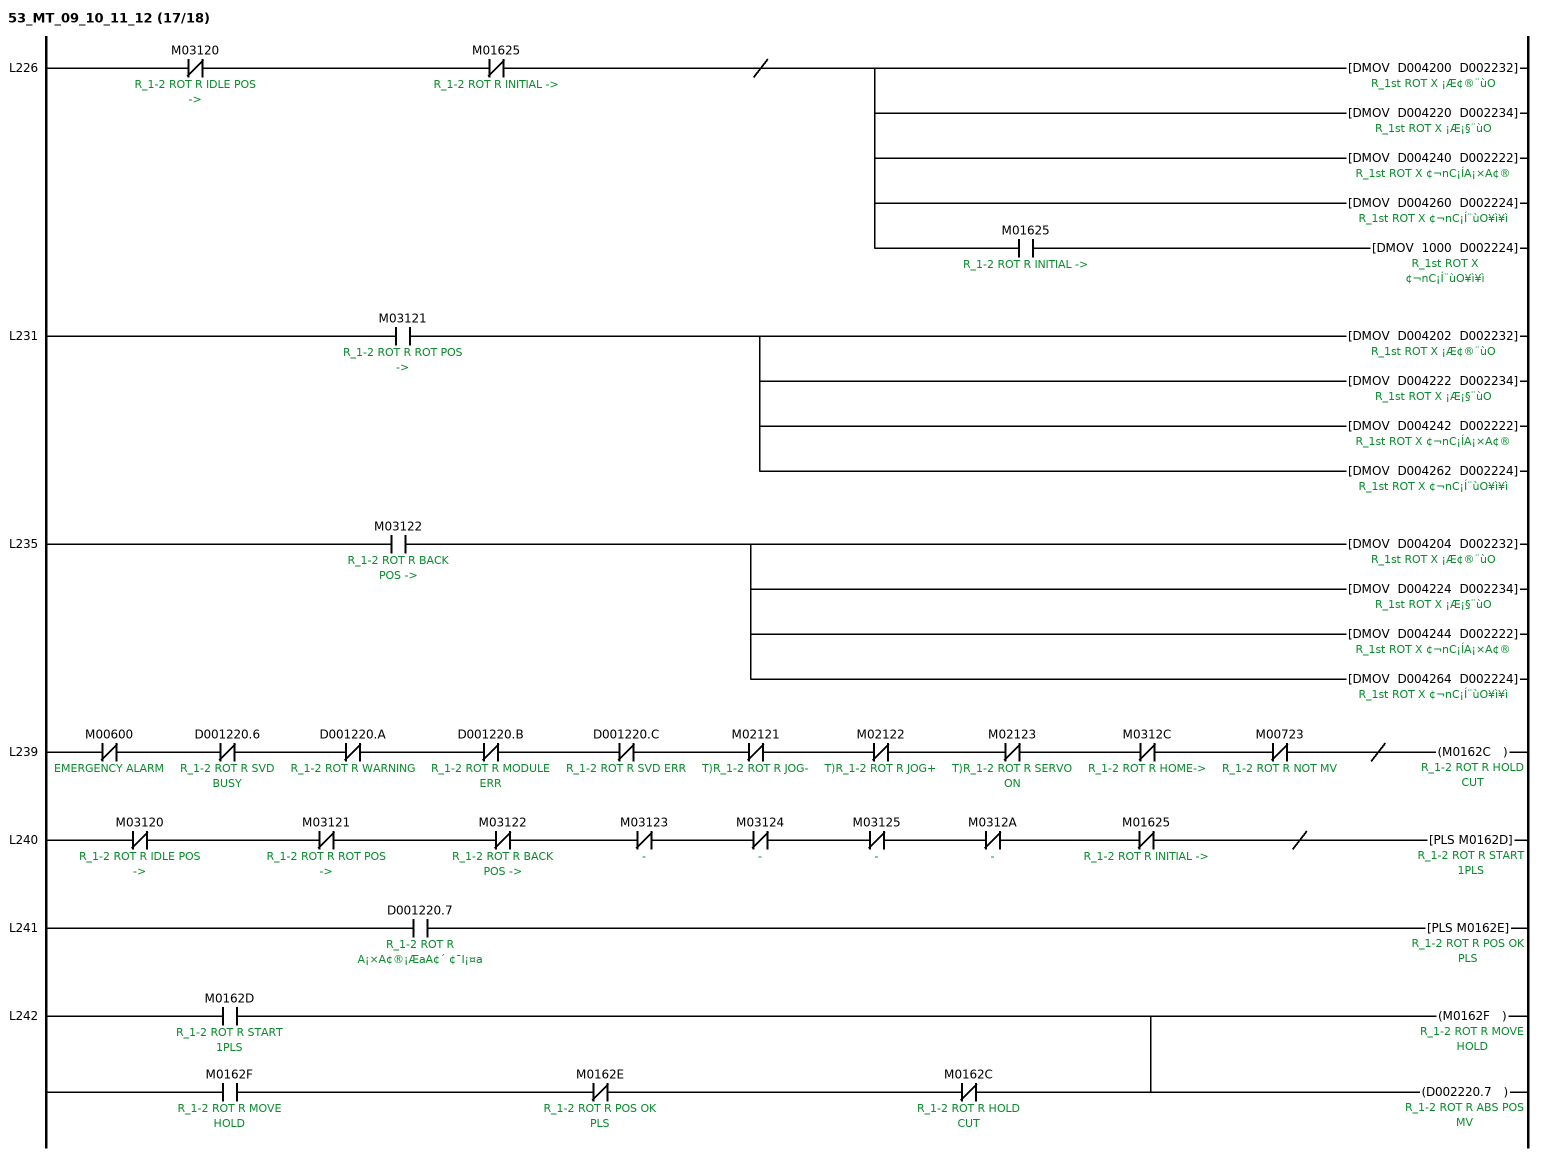
; L226
LOAD NOT  M03120	// R_1-2 ROT R IDLE POS ->
AND NOT   M01625	// R_1-2 ROT R INITIAL ->
NOT
DMOV      D004200 D002232	// R_1st ROT X ¡Æ¢®¨ùO
DMOV      D004220 D002234	// R_1st ROT X ¡Æ¡§¨ùO
DMOV      D004240 D002222	// R_1st ROT X ¢¬nC¡ÍA¡×A¢®
DMOV      D004260 D002224	// R_1st ROT X ¢¬nC¡Í¨ùO¥ì¥ì
AND       M01625	// R_1-2 ROT R INITIAL ->
DMOV      1000 D002224	// R_1st ROT X ¢¬nC¡Í¨ùO¥ì¥ì
; L231
LOAD      M03121	// R_1-2 ROT R ROT POS ->
DMOV      D004202 D002232	// R_1st ROT X ¡Æ¢®¨ùO
DMOV      D004222 D002234	// R_1st ROT X ¡Æ¡§¨ùO
DMOV      D004242 D002222	// R_1st ROT X ¢¬nC¡ÍA¡×A¢®
DMOV      D004262 D002224	// R_1st ROT X ¢¬nC¡Í¨ùO¥ì¥ì
; L235
LOAD      M03122	// R_1-2 ROT R BACK POS ->
DMOV      D004204 D002232	// R_1st ROT X ¡Æ¢®¨ùO
DMOV      D004224 D002234	// R_1st ROT X ¡Æ¡§¨ùO
DMOV      D004244 D002222	// R_1st ROT X ¢¬nC¡ÍA¡×A¢®
DMOV      D004264 D002224	// R_1st ROT X ¢¬nC¡Í¨ùO¥ì¥ì
; L239
LOAD NOT  M00600	// EMERGENCY ALARM
AND NOT   D001220.6	// R_1-2 ROT R SVD BUSY
AND NOT   D001220.A	// R_1-2 ROT R WARNING
AND NOT   D001220.B	// R_1-2 ROT R MODULE ERR
AND NOT   D001220.C	// R_1-2 ROT R SVD ERR
AND NOT   M02121	// T)R_1-2 ROT R JOG-
AND NOT   M02122	// T)R_1-2 ROT R JOG+
AND NOT   M02123	// T)R_1-2 ROT R SERVO ON
AND NOT   M0312C	// R_1-2 ROT R HOME->
AND NOT   M00723	// R_1-2 ROT R NOT MV
NOT
OUT       M0162C	// R_1-2 ROT R HOLD CUT
; L240
LOAD NOT  M03120	// R_1-2 ROT R IDLE POS ->
AND NOT   M03121	// R_1-2 ROT R ROT POS ->
AND NOT   M03122	// R_1-2 ROT R BACK POS ->
AND NOT   M03123	// -
AND NOT   M03124	// -
AND NOT   M03125	// -
AND NOT   M0312A	// -
AND NOT   M01625	// R_1-2 ROT R INITIAL ->
NOT
OUTP      M0162D	// R_1-2 ROT R START 1PLS
; L241
LOAD      D001220.7	// R_1-2 ROT R A¡×A¢®¡ÆaA¢´ ¢¯I¡¤a
OUTP      M0162E	// R_1-2 ROT R POS OK PLS
; L242
LOAD      M0162D	// R_1-2 ROT R START 1PLS
LOAD      M0162F	// R_1-2 ROT R MOVE HOLD
AND NOT   M0162E	// R_1-2 ROT R POS OK PLS
AND NOT   M0162C	// R_1-2 ROT R HOLD CUT
OR LOAD
OUT       M0162F	// R_1-2 ROT R MOVE HOLD
OUT       D002220.7	// R_1-2 ROT R ABS POS MV

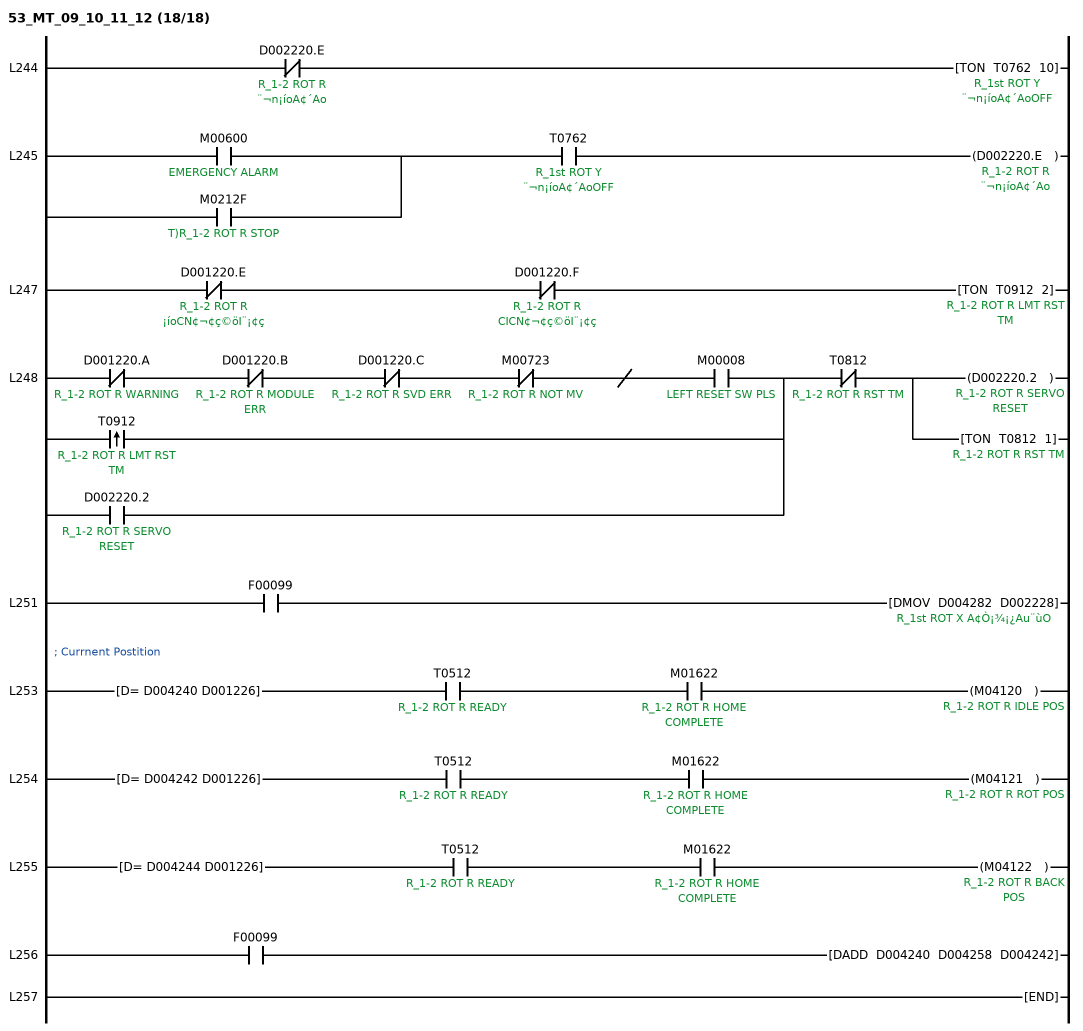
; L244
LOAD NOT  D002220.E	// R_1-2 ROT R ¨¬n¡íoA¢´Ao
TON       T0762 10	// R_1st ROT Y ¨¬n¡íoA¢´AoOFF
; L245
LOAD      M00600	// EMERGENCY ALARM
OR        M0212F	// T)R_1-2 ROT R STOP
AND       T0762	// R_1st ROT Y ¨¬n¡íoA¢´AoOFF
OUT       D002220.E	// R_1-2 ROT R ¨¬n¡íoA¢´Ao
; L247
LOAD NOT  D001220.E	// R_1-2 ROT R ¡íoCN¢¬¢ç©öI¨¡¢ç
AND NOT   D001220.F	// R_1-2 ROT R CICN¢¬¢ç©öI¨¡¢ç
TON       T0912 2	// R_1-2 ROT R LMT RST TM
; L248
LOAD NOT  D001220.A	// R_1-2 ROT R WARNING
AND NOT   D001220.B	// R_1-2 ROT R MODULE ERR
AND NOT   D001220.C	// R_1-2 ROT R SVD ERR
AND NOT   M00723	// R_1-2 ROT R NOT MV
NOT
AND       M00008	// LEFT RESET SW PLS
ORP       T0912	// R_1-2 ROT R LMT RST TM
OR        D002220.2	// R_1-2 ROT R SERVO RESET
AND NOT   T0812	// R_1-2 ROT R RST TM
OUT       D002220.2	// R_1-2 ROT R SERVO RESET
TON       T0812 1	// R_1-2 ROT R RST TM
; L251
LOAD      F00099
DMOV      D004282 D002228	// R_1st ROT X A¢Ò¡¾¡¿Au¨ùO
// Currnent Postition
; L253
LOADD=    D004240 D001226
AND       T0512	// R_1-2 ROT R READY
AND       M01622	// R_1-2 ROT R HOME COMPLETE
OUT       M04120	// R_1-2 ROT R IDLE POS
; L254
LOADD=    D004242 D001226
AND       T0512	// R_1-2 ROT R READY
AND       M01622	// R_1-2 ROT R HOME COMPLETE
OUT       M04121	// R_1-2 ROT R ROT POS
; L255
LOADD=    D004244 D001226
AND       T0512	// R_1-2 ROT R READY
AND       M01622	// R_1-2 ROT R HOME COMPLETE
OUT       M04122	// R_1-2 ROT R BACK POS
; L256
LOAD      F00099
DADD      D004240 D004258 D004242
; L257
END

PROGRAM 54_MT_13_14_15_16 (task: ¨ö¨¬A¥ì CA¡¤I¡¾¡¿¡¤¡Í)

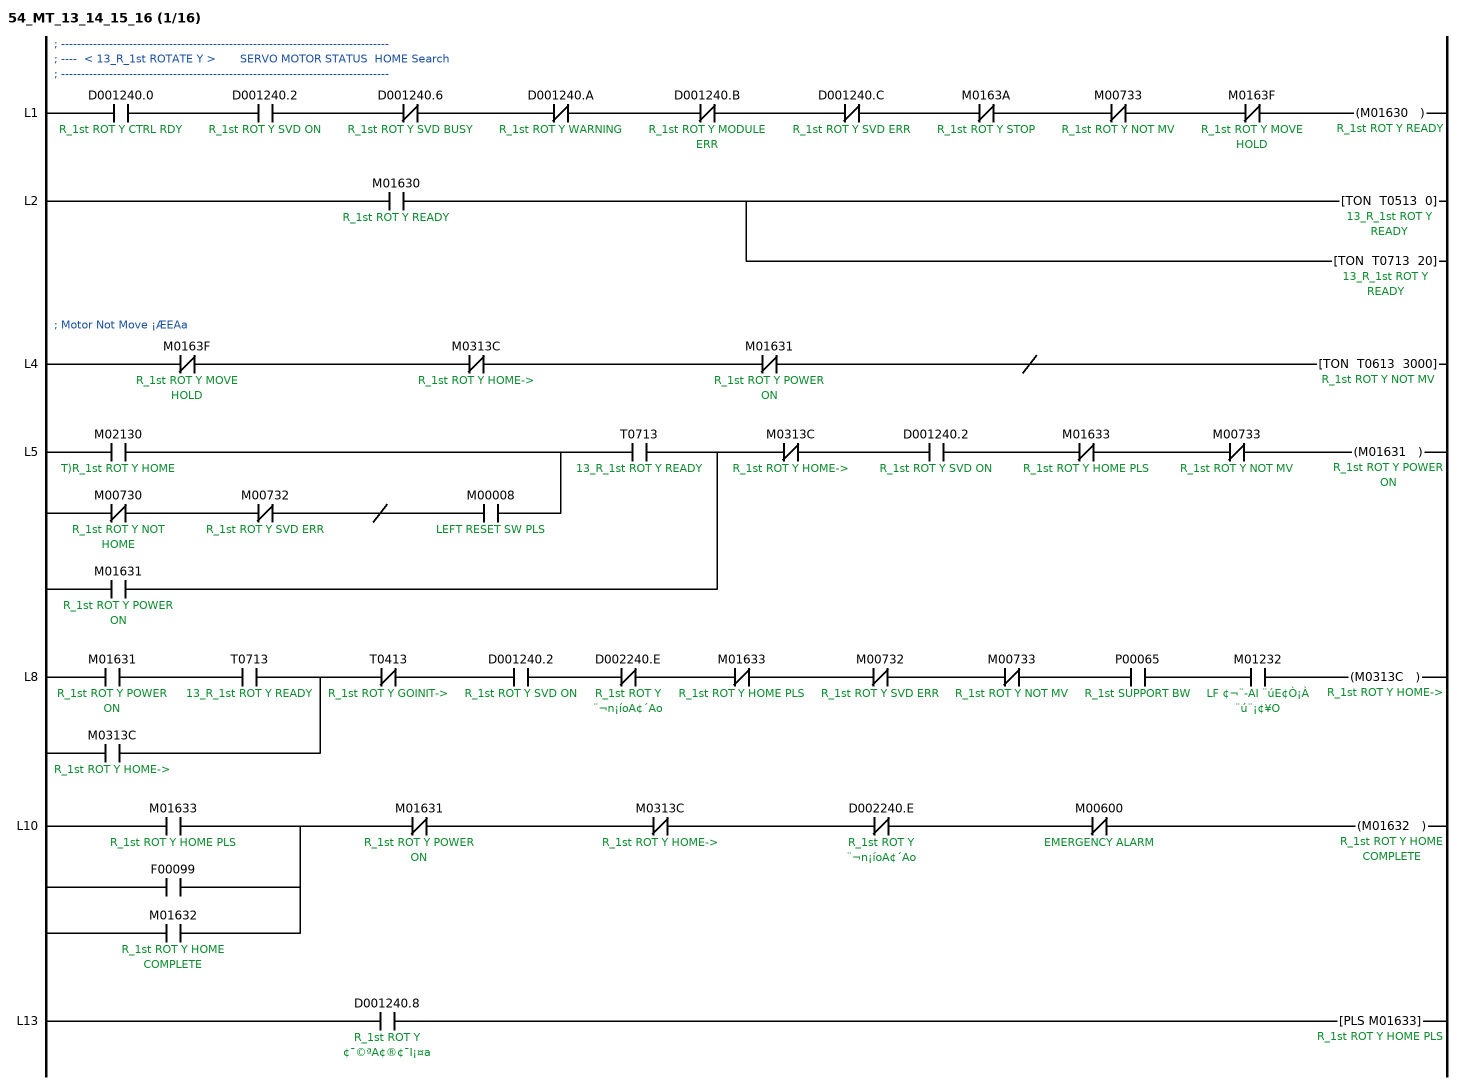
// ----------------------------------------------------------------------------------
// 
// ----  < 13_R_1st ROTATE Y >       SERVO MOTOR STATUS  HOME Search
// 
// ----------------------------------------------------------------------------------
; L1
LOAD      D001240.0	// R_1st ROT Y CTRL RDY
AND       D001240.2	// R_1st ROT Y SVD ON
AND NOT   D001240.6	// R_1st ROT Y SVD BUSY
AND NOT   D001240.A	// R_1st ROT Y WARNING
AND NOT   D001240.B	// R_1st ROT Y MODULE ERR
AND NOT   D001240.C	// R_1st ROT Y SVD ERR
AND NOT   M0163A	// R_1st ROT Y STOP
AND NOT   M00733	// R_1st ROT Y NOT MV
AND NOT   M0163F	// R_1st ROT Y MOVE HOLD
OUT       M01630	// R_1st ROT Y READY
; L2
LOAD      M01630	// R_1st ROT Y READY
TON       T0513 0	// 13_R_1st ROT Y READY
TON       T0713 20	// 13_R_1st ROT Y READY
; L4
LOAD NOT  M0163F	// R_1st ROT Y MOVE HOLD
AND NOT   M0313C	// R_1st ROT Y HOME->
AND NOT   M01631	// R_1st ROT Y POWER ON
NOT
TON       T0613 3000	// R_1st ROT Y NOT MV
// output comment: Motor Not Move ¡ÆEAa
; L5
LOAD      M02130	// T)R_1st ROT Y HOME
LOAD NOT  M00730	// R_1st ROT Y NOT HOME
AND NOT   M00732	// R_1st ROT Y SVD ERR
NOT
AND       M00008	// LEFT RESET SW PLS
OR LOAD
AND       T0713	// 13_R_1st ROT Y READY
OR        M01631	// R_1st ROT Y POWER ON
AND NOT   M0313C	// R_1st ROT Y HOME->
AND       D001240.2	// R_1st ROT Y SVD ON
AND NOT   M01633	// R_1st ROT Y HOME PLS
AND NOT   M00733	// R_1st ROT Y NOT MV
OUT       M01631	// R_1st ROT Y POWER ON
; L8
LOAD      M01631	// R_1st ROT Y POWER ON
AND       T0713	// 13_R_1st ROT Y READY
OR        M0313C	// R_1st ROT Y HOME->
AND NOT   T0413	// R_1st ROT Y GOINIT->
AND       D001240.2	// R_1st ROT Y SVD ON
AND NOT   D002240.E	// R_1st ROT Y ¨¬n¡íoA¢´Ao
AND NOT   M01633	// R_1st ROT Y HOME PLS
AND NOT   M00732	// R_1st ROT Y SVD ERR
AND NOT   M00733	// R_1st ROT Y NOT MV
AND       P00065	// R_1st SUPPORT BW
AND       M01232	// LF ¢¬¨­AI ¨úE¢Ò¡À ¨ú¨¡¢¥O
OUT       M0313C	// R_1st ROT Y HOME->
; L10
LOAD      M01633	// R_1st ROT Y HOME PLS
OR        F00099
OR        M01632	// R_1st ROT Y HOME COMPLETE
AND NOT   M01631	// R_1st ROT Y POWER ON
AND NOT   M0313C	// R_1st ROT Y HOME->
AND NOT   D002240.E	// R_1st ROT Y ¨¬n¡íoA¢´Ao
AND NOT   M00600	// EMERGENCY ALARM
OUT       M01632	// R_1st ROT Y HOME COMPLETE
; L13
LOAD      D001240.8	// R_1st ROT Y ¢¯©ªA¢®¢¯I¡¤a
OUTP      M01633	// R_1st ROT Y HOME PLS

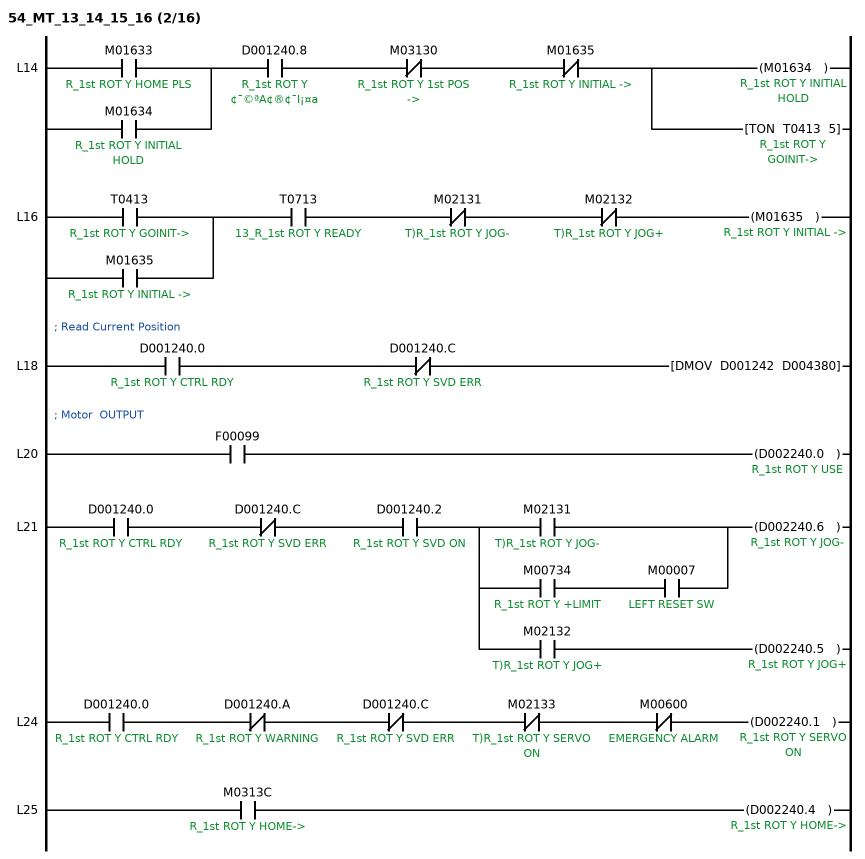
; L14
LOAD      M01633	// R_1st ROT Y HOME PLS
OR        M01634	// R_1st ROT Y INITIAL HOLD
AND       D001240.8	// R_1st ROT Y ¢¯©ªA¢®¢¯I¡¤a
AND NOT   M03130	// R_1st ROT Y 1st POS ->
AND NOT   M01635	// R_1st ROT Y INITIAL ->
OUT       M01634	// R_1st ROT Y INITIAL HOLD
TON       T0413 5	// R_1st ROT Y GOINIT->
; L16
LOAD      T0413	// R_1st ROT Y GOINIT->
OR        M01635	// R_1st ROT Y INITIAL ->
AND       T0713	// 13_R_1st ROT Y READY
AND NOT   M02131	// T)R_1st ROT Y JOG-
AND NOT   M02132	// T)R_1st ROT Y JOG+
OUT       M01635	// R_1st ROT Y INITIAL ->
; L18
LOAD      D001240.0	// R_1st ROT Y CTRL RDY
AND NOT   D001240.C	// R_1st ROT Y SVD ERR
DMOV      D001242 D004380
// output comment: Read Current Position
//  Motor  OUTPUT
; L20
LOAD      F00099
OUT       D002240.0	// R_1st ROT Y USE
; L21
LOAD      D001240.0	// R_1st ROT Y CTRL RDY
AND NOT   D001240.C	// R_1st ROT Y SVD ERR
AND       D001240.2	// R_1st ROT Y SVD ON
MPUSH
LOAD      M02131	// T)R_1st ROT Y JOG-
LOAD      M00734	// R_1st ROT Y +LIMIT
AND       M00007	// LEFT RESET SW
OR LOAD
AND LOAD
OUT       D002240.6	// R_1st ROT Y JOG-
MPOP
AND       M02132	// T)R_1st ROT Y JOG+
OUT       D002240.5	// R_1st ROT Y JOG+
; L24
LOAD      D001240.0	// R_1st ROT Y CTRL RDY
AND NOT   D001240.A	// R_1st ROT Y WARNING
AND NOT   D001240.C	// R_1st ROT Y SVD ERR
AND NOT   M02133	// T)R_1st ROT Y SERVO ON
AND NOT   M00600	// EMERGENCY ALARM
OUT       D002240.1	// R_1st ROT Y SERVO ON
; L25
LOAD      M0313C	// R_1st ROT Y HOME->
OUT       D002240.4	// R_1st ROT Y HOME->

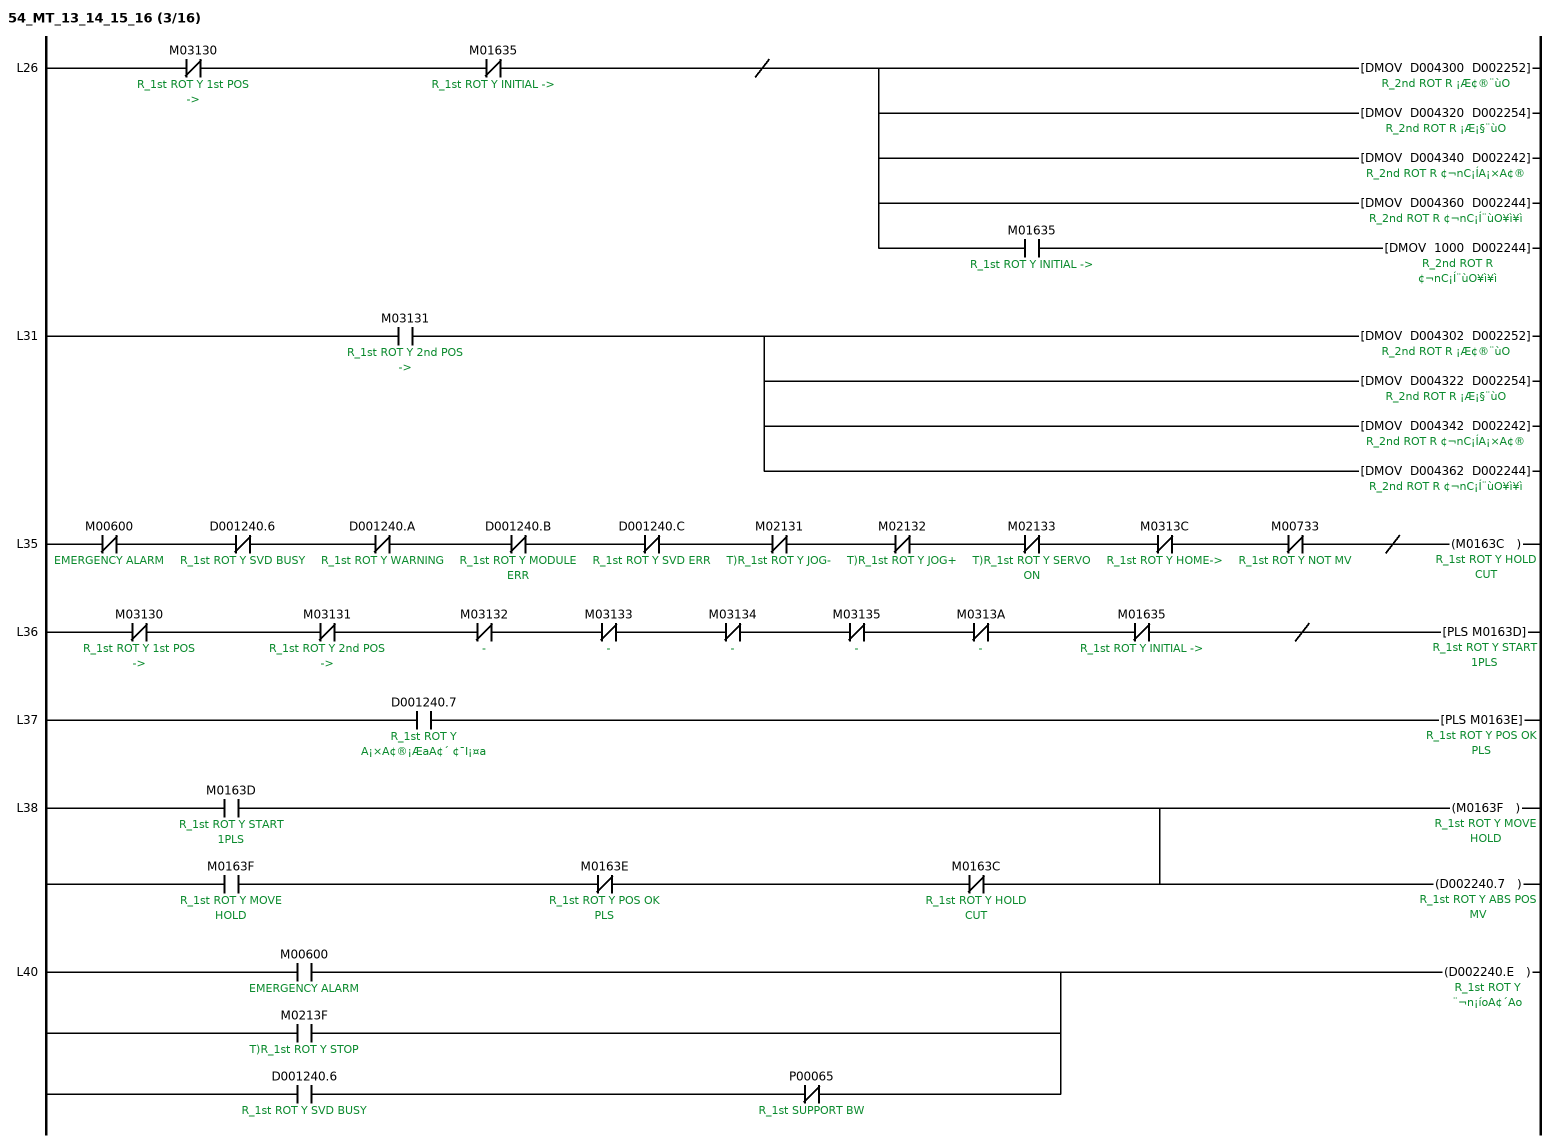
; L26
LOAD NOT  M03130	// R_1st ROT Y 1st POS ->
AND NOT   M01635	// R_1st ROT Y INITIAL ->
NOT
DMOV      D004300 D002252	// R_2nd ROT R ¡Æ¢®¨ùO
DMOV      D004320 D002254	// R_2nd ROT R ¡Æ¡§¨ùO
DMOV      D004340 D002242	// R_2nd ROT R ¢¬nC¡ÍA¡×A¢®
DMOV      D004360 D002244	// R_2nd ROT R ¢¬nC¡Í¨ùO¥ì¥ì
AND       M01635	// R_1st ROT Y INITIAL ->
DMOV      1000 D002244	// R_2nd ROT R ¢¬nC¡Í¨ùO¥ì¥ì
; L31
LOAD      M03131	// R_1st ROT Y 2nd POS ->
DMOV      D004302 D002252	// R_2nd ROT R ¡Æ¢®¨ùO
DMOV      D004322 D002254	// R_2nd ROT R ¡Æ¡§¨ùO
DMOV      D004342 D002242	// R_2nd ROT R ¢¬nC¡ÍA¡×A¢®
DMOV      D004362 D002244	// R_2nd ROT R ¢¬nC¡Í¨ùO¥ì¥ì
; L35
LOAD NOT  M00600	// EMERGENCY ALARM
AND NOT   D001240.6	// R_1st ROT Y SVD BUSY
AND NOT   D001240.A	// R_1st ROT Y WARNING
AND NOT   D001240.B	// R_1st ROT Y MODULE ERR
AND NOT   D001240.C	// R_1st ROT Y SVD ERR
AND NOT   M02131	// T)R_1st ROT Y JOG-
AND NOT   M02132	// T)R_1st ROT Y JOG+
AND NOT   M02133	// T)R_1st ROT Y SERVO ON
AND NOT   M0313C	// R_1st ROT Y HOME->
AND NOT   M00733	// R_1st ROT Y NOT MV
NOT
OUT       M0163C	// R_1st ROT Y HOLD CUT
; L36
LOAD NOT  M03130	// R_1st ROT Y 1st POS ->
AND NOT   M03131	// R_1st ROT Y 2nd POS ->
AND NOT   M03132	// -
AND NOT   M03133	// -
AND NOT   M03134	// -
AND NOT   M03135	// -
AND NOT   M0313A	// -
AND NOT   M01635	// R_1st ROT Y INITIAL ->
NOT
OUTP      M0163D	// R_1st ROT Y START 1PLS
; L37
LOAD      D001240.7	// R_1st ROT Y A¡×A¢®¡ÆaA¢´ ¢¯I¡¤a
OUTP      M0163E	// R_1st ROT Y POS OK PLS
; L38
LOAD      M0163D	// R_1st ROT Y START 1PLS
LOAD      M0163F	// R_1st ROT Y MOVE HOLD
AND NOT   M0163E	// R_1st ROT Y POS OK PLS
AND NOT   M0163C	// R_1st ROT Y HOLD CUT
OR LOAD
OUT       M0163F	// R_1st ROT Y MOVE HOLD
OUT       D002240.7	// R_1st ROT Y ABS POS MV
; L40
LOAD      M00600	// EMERGENCY ALARM
OR        M0213F	// T)R_1st ROT Y STOP
LOAD      D001240.6	// R_1st ROT Y SVD BUSY
AND NOT   P00065	// R_1st SUPPORT BW
OR LOAD
OUT       D002240.E	// R_1st ROT Y ¨¬n¡íoA¢´Ao

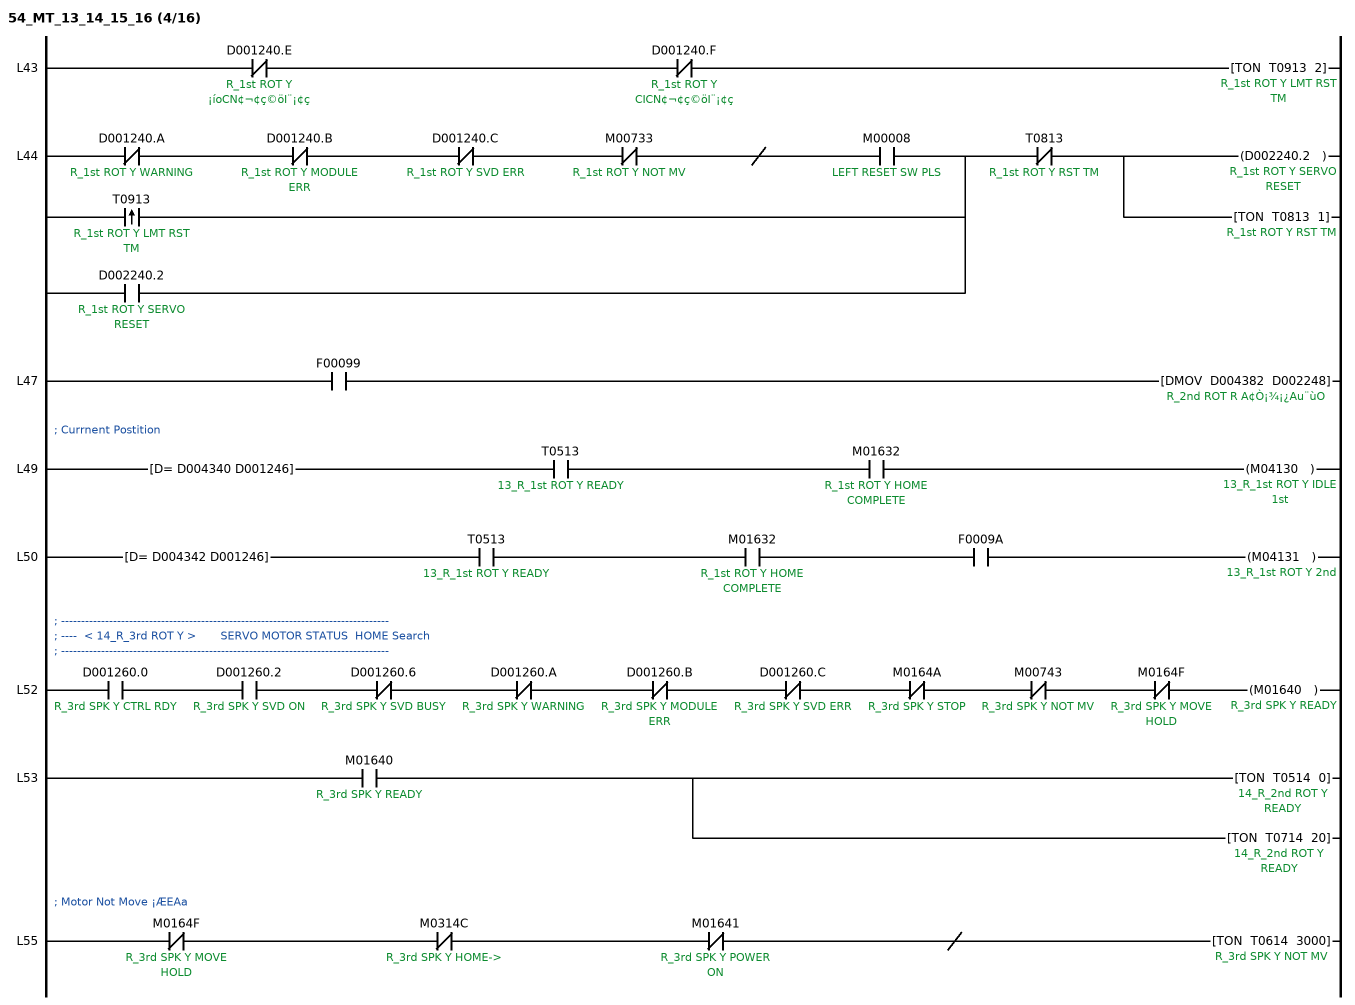
; L43
LOAD NOT  D001240.E	// R_1st ROT Y ¡íoCN¢¬¢ç©öI¨¡¢ç
AND NOT   D001240.F	// R_1st ROT Y CICN¢¬¢ç©öI¨¡¢ç
TON       T0913 2	// R_1st ROT Y LMT RST TM
; L44
LOAD NOT  D001240.A	// R_1st ROT Y WARNING
AND NOT   D001240.B	// R_1st ROT Y MODULE ERR
AND NOT   D001240.C	// R_1st ROT Y SVD ERR
AND NOT   M00733	// R_1st ROT Y NOT MV
NOT
AND       M00008	// LEFT RESET SW PLS
ORP       T0913	// R_1st ROT Y LMT RST TM
OR        D002240.2	// R_1st ROT Y SERVO RESET
AND NOT   T0813	// R_1st ROT Y RST TM
OUT       D002240.2	// R_1st ROT Y SERVO RESET
TON       T0813 1	// R_1st ROT Y RST TM
; L47
LOAD      F00099
DMOV      D004382 D002248	// R_2nd ROT R A¢Ò¡¾¡¿Au¨ùO
// Currnent Postition
; L49
LOADD=    D004340 D001246
AND       T0513	// 13_R_1st ROT Y READY
AND       M01632	// R_1st ROT Y HOME COMPLETE
OUT       M04130	// 13_R_1st ROT Y IDLE 1st
; L50
LOADD=    D004342 D001246
AND       T0513	// 13_R_1st ROT Y READY
AND       M01632	// R_1st ROT Y HOME COMPLETE
AND       F0009A
OUT       M04131	// 13_R_1st ROT Y 2nd
// ----------------------------------------------------------------------------------
// 
// ----  < 14_R_3rd ROT Y >       SERVO MOTOR STATUS  HOME Search
// 
// ----------------------------------------------------------------------------------
; L52
LOAD      D001260.0	// R_3rd SPK Y CTRL RDY
AND       D001260.2	// R_3rd SPK Y SVD ON
AND NOT   D001260.6	// R_3rd SPK Y SVD BUSY
AND NOT   D001260.A	// R_3rd SPK Y WARNING
AND NOT   D001260.B	// R_3rd SPK Y MODULE ERR
AND NOT   D001260.C	// R_3rd SPK Y SVD ERR
AND NOT   M0164A	// R_3rd SPK Y STOP
AND NOT   M00743	// R_3rd SPK Y NOT MV
AND NOT   M0164F	// R_3rd SPK Y MOVE HOLD
OUT       M01640	// R_3rd SPK Y READY
; L53
LOAD      M01640	// R_3rd SPK Y READY
TON       T0514 0	// 14_R_2nd ROT Y READY
TON       T0714 20	// 14_R_2nd ROT Y READY
; L55
LOAD NOT  M0164F	// R_3rd SPK Y MOVE HOLD
AND NOT   M0314C	// R_3rd SPK Y HOME->
AND NOT   M01641	// R_3rd SPK Y POWER ON
NOT
TON       T0614 3000	// R_3rd SPK Y NOT MV
// output comment: Motor Not Move ¡ÆEAa

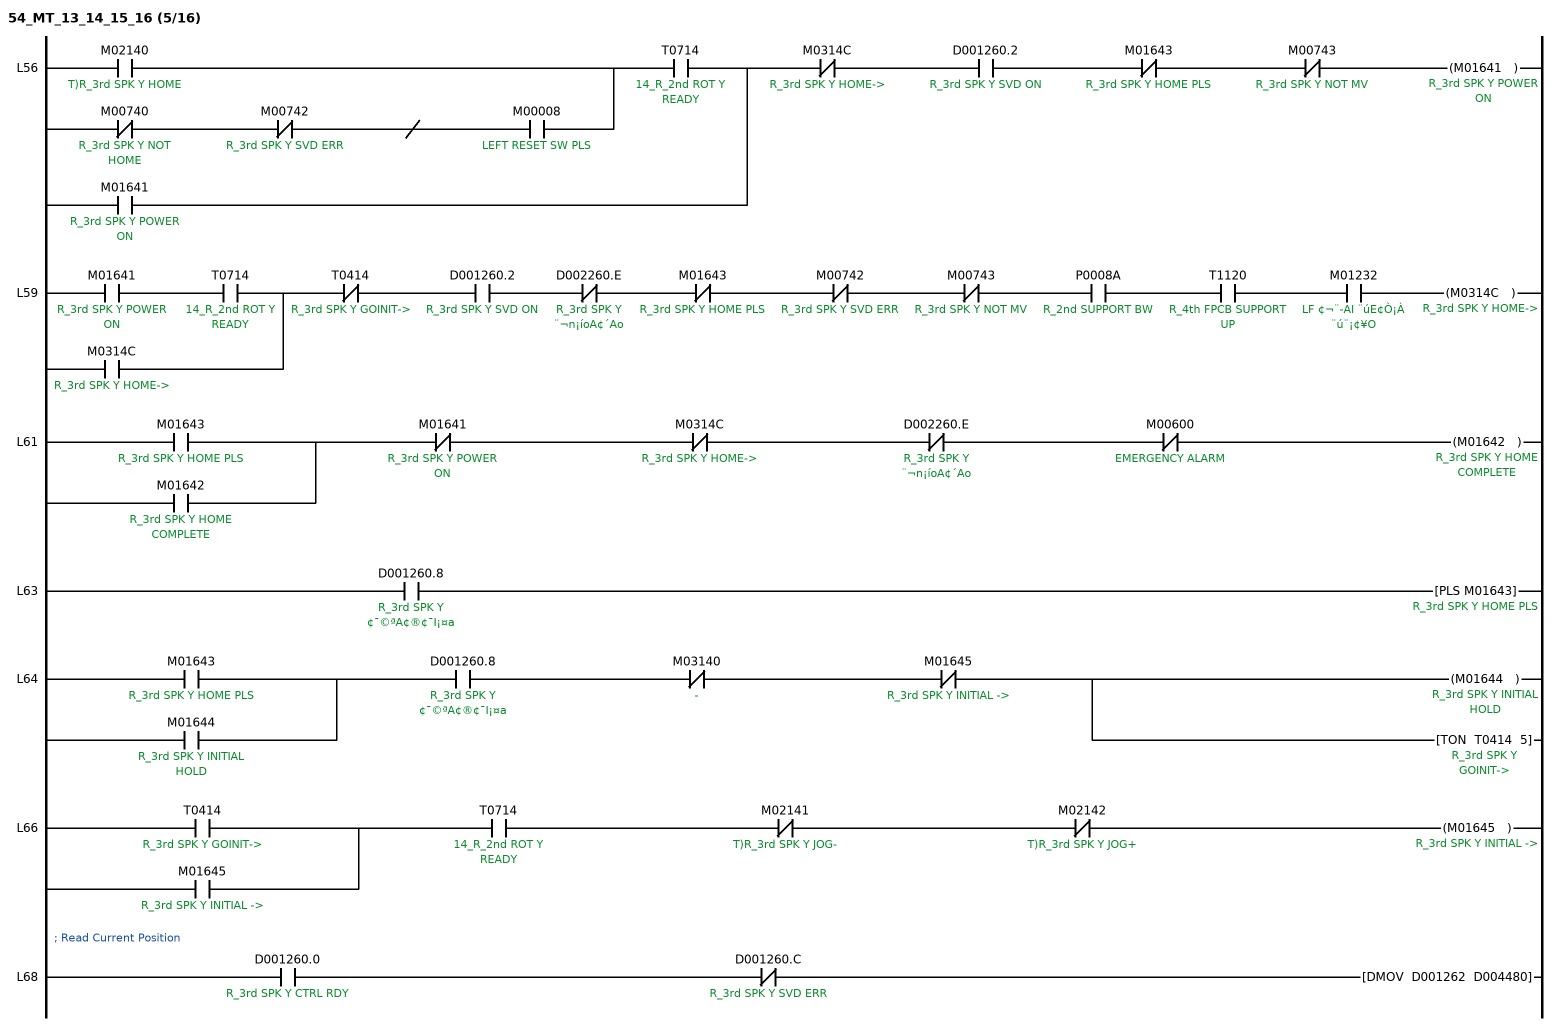
; L56
LOAD      M02140	// T)R_3rd SPK Y HOME
LOAD NOT  M00740	// R_3rd SPK Y NOT HOME
AND NOT   M00742	// R_3rd SPK Y SVD ERR
NOT
AND       M00008	// LEFT RESET SW PLS
OR LOAD
AND       T0714	// 14_R_2nd ROT Y READY
OR        M01641	// R_3rd SPK Y POWER ON
AND NOT   M0314C	// R_3rd SPK Y HOME->
AND       D001260.2	// R_3rd SPK Y SVD ON
AND NOT   M01643	// R_3rd SPK Y HOME PLS
AND NOT   M00743	// R_3rd SPK Y NOT MV
OUT       M01641	// R_3rd SPK Y POWER ON
; L59
LOAD      M01641	// R_3rd SPK Y POWER ON
AND       T0714	// 14_R_2nd ROT Y READY
OR        M0314C	// R_3rd SPK Y HOME->
AND NOT   T0414	// R_3rd SPK Y GOINIT->
AND       D001260.2	// R_3rd SPK Y SVD ON
AND NOT   D002260.E	// R_3rd SPK Y ¨¬n¡íoA¢´Ao
AND NOT   M01643	// R_3rd SPK Y HOME PLS
AND NOT   M00742	// R_3rd SPK Y SVD ERR
AND NOT   M00743	// R_3rd SPK Y NOT MV
AND       P0008A	// R_2nd SUPPORT BW
AND       T1120	// R_4th FPCB SUPPORT UP
AND       M01232	// LF ¢¬¨­AI ¨úE¢Ò¡À ¨ú¨¡¢¥O
OUT       M0314C	// R_3rd SPK Y HOME->
; L61
LOAD      M01643	// R_3rd SPK Y HOME PLS
OR        M01642	// R_3rd SPK Y HOME COMPLETE
AND NOT   M01641	// R_3rd SPK Y POWER ON
AND NOT   M0314C	// R_3rd SPK Y HOME->
AND NOT   D002260.E	// R_3rd SPK Y ¨¬n¡íoA¢´Ao
AND NOT   M00600	// EMERGENCY ALARM
OUT       M01642	// R_3rd SPK Y HOME COMPLETE
; L63
LOAD      D001260.8	// R_3rd SPK Y ¢¯©ªA¢®¢¯I¡¤a
OUTP      M01643	// R_3rd SPK Y HOME PLS
; L64
LOAD      M01643	// R_3rd SPK Y HOME PLS
OR        M01644	// R_3rd SPK Y INITIAL HOLD
AND       D001260.8	// R_3rd SPK Y ¢¯©ªA¢®¢¯I¡¤a
AND NOT   M03140	// -
AND NOT   M01645	// R_3rd SPK Y INITIAL ->
OUT       M01644	// R_3rd SPK Y INITIAL HOLD
TON       T0414 5	// R_3rd SPK Y GOINIT->
; L66
LOAD      T0414	// R_3rd SPK Y GOINIT->
OR        M01645	// R_3rd SPK Y INITIAL ->
AND       T0714	// 14_R_2nd ROT Y READY
AND NOT   M02141	// T)R_3rd SPK Y JOG-
AND NOT   M02142	// T)R_3rd SPK Y JOG+
OUT       M01645	// R_3rd SPK Y INITIAL ->
; L68
LOAD      D001260.0	// R_3rd SPK Y CTRL RDY
AND NOT   D001260.C	// R_3rd SPK Y SVD ERR
DMOV      D001262 D004480
// output comment: Read Current Position

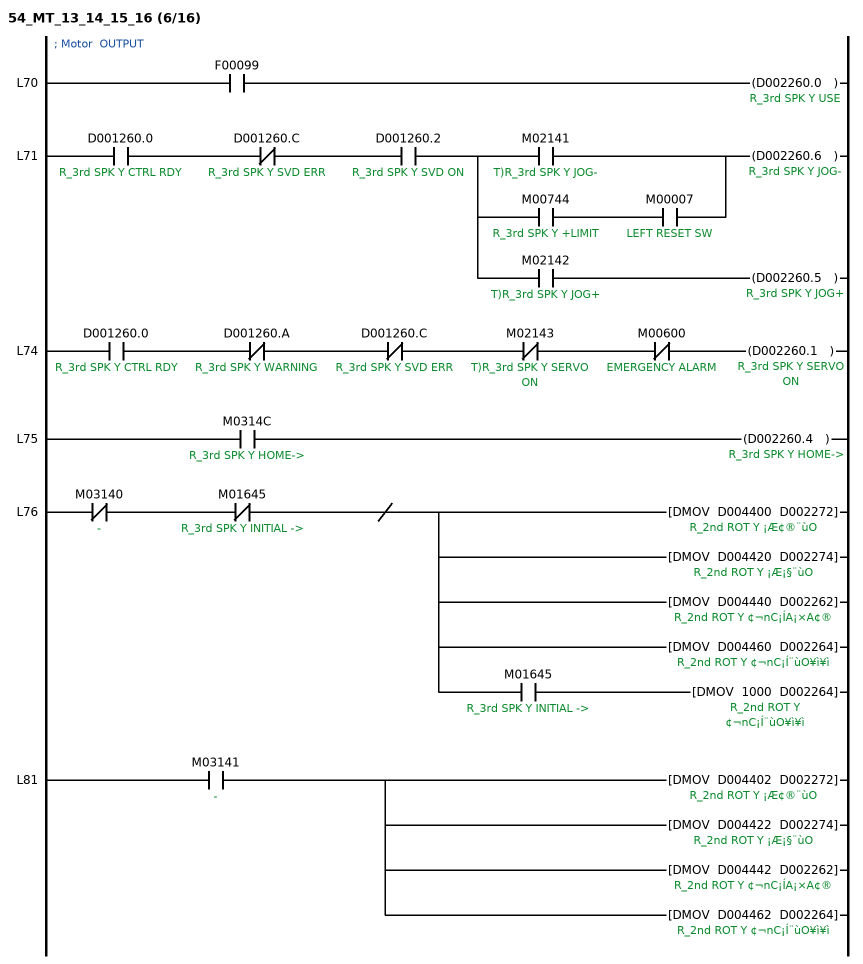
//  Motor  OUTPUT
; L70
LOAD      F00099
OUT       D002260.0	// R_3rd SPK Y USE
; L71
LOAD      D001260.0	// R_3rd SPK Y CTRL RDY
AND NOT   D001260.C	// R_3rd SPK Y SVD ERR
AND       D001260.2	// R_3rd SPK Y SVD ON
MPUSH
LOAD      M02141	// T)R_3rd SPK Y JOG-
LOAD      M00744	// R_3rd SPK Y +LIMIT
AND       M00007	// LEFT RESET SW
OR LOAD
AND LOAD
OUT       D002260.6	// R_3rd SPK Y JOG-
MPOP
AND       M02142	// T)R_3rd SPK Y JOG+
OUT       D002260.5	// R_3rd SPK Y JOG+
; L74
LOAD      D001260.0	// R_3rd SPK Y CTRL RDY
AND NOT   D001260.A	// R_3rd SPK Y WARNING
AND NOT   D001260.C	// R_3rd SPK Y SVD ERR
AND NOT   M02143	// T)R_3rd SPK Y SERVO ON
AND NOT   M00600	// EMERGENCY ALARM
OUT       D002260.1	// R_3rd SPK Y SERVO ON
; L75
LOAD      M0314C	// R_3rd SPK Y HOME->
OUT       D002260.4	// R_3rd SPK Y HOME->
; L76
LOAD NOT  M03140	// -
AND NOT   M01645	// R_3rd SPK Y INITIAL ->
NOT
DMOV      D004400 D002272	// R_2nd ROT Y ¡Æ¢®¨ùO
DMOV      D004420 D002274	// R_2nd ROT Y ¡Æ¡§¨ùO
DMOV      D004440 D002262	// R_2nd ROT Y ¢¬nC¡ÍA¡×A¢®
DMOV      D004460 D002264	// R_2nd ROT Y ¢¬nC¡Í¨ùO¥ì¥ì
AND       M01645	// R_3rd SPK Y INITIAL ->
DMOV      1000 D002264	// R_2nd ROT Y ¢¬nC¡Í¨ùO¥ì¥ì
; L81
LOAD      M03141	// -
DMOV      D004402 D002272	// R_2nd ROT Y ¡Æ¢®¨ùO
DMOV      D004422 D002274	// R_2nd ROT Y ¡Æ¡§¨ùO
DMOV      D004442 D002262	// R_2nd ROT Y ¢¬nC¡ÍA¡×A¢®
DMOV      D004462 D002264	// R_2nd ROT Y ¢¬nC¡Í¨ùO¥ì¥ì

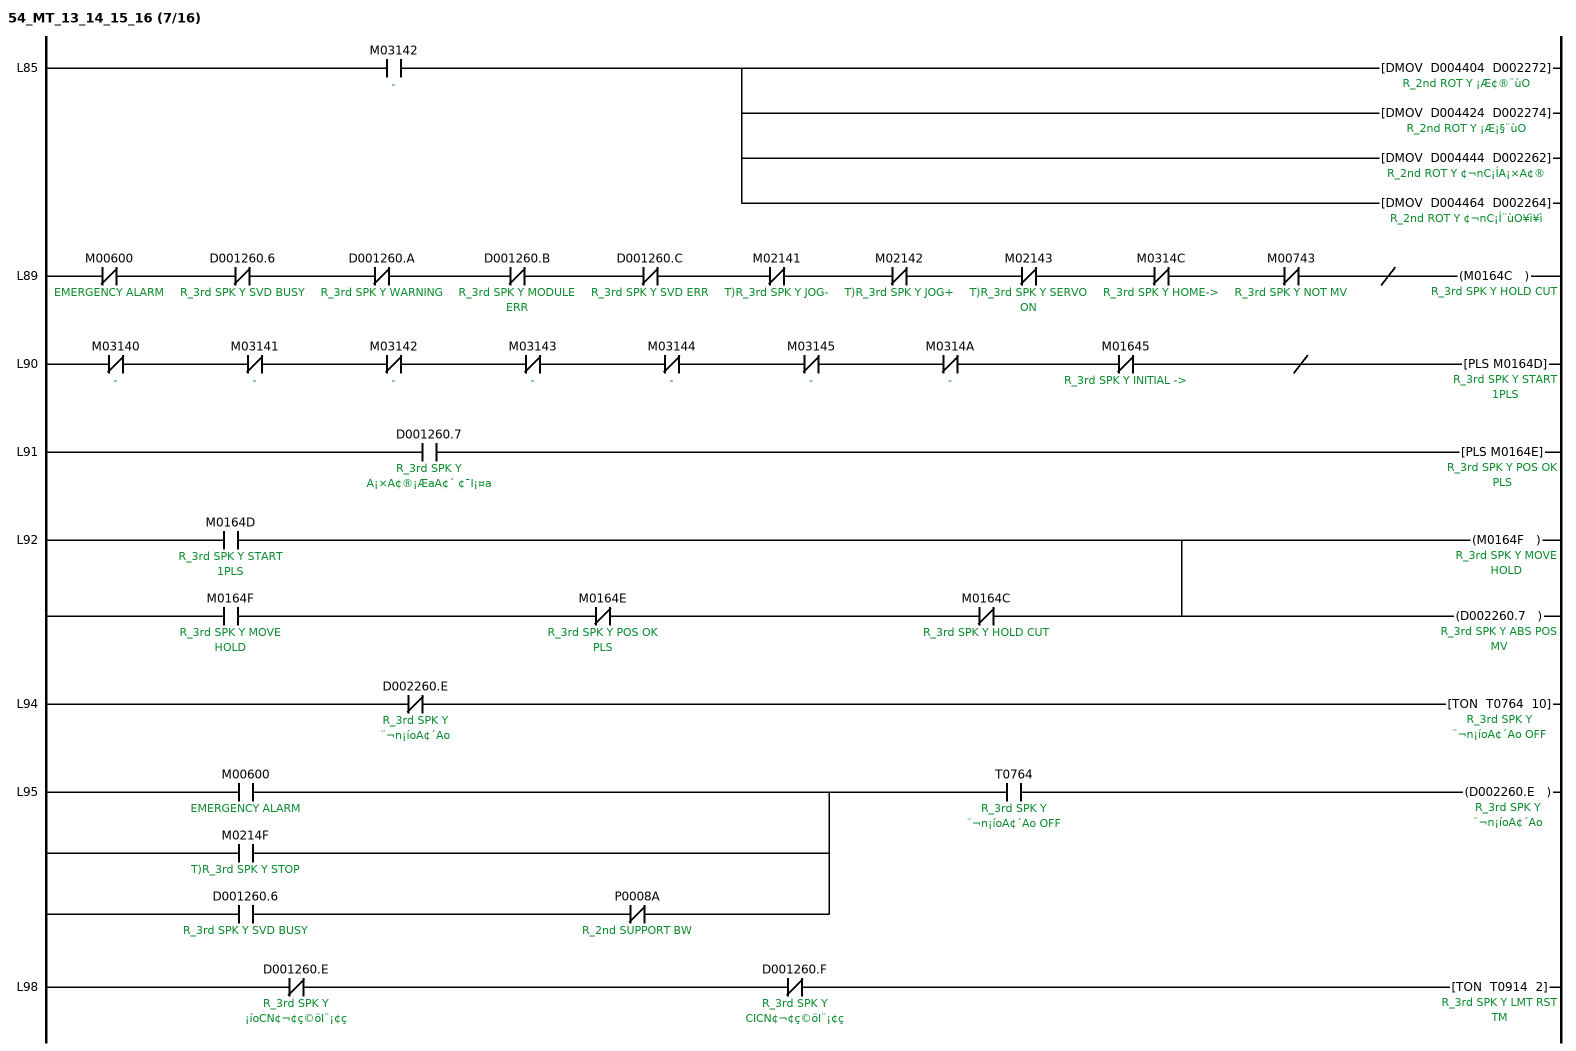
; L85
LOAD      M03142	// -
DMOV      D004404 D002272	// R_2nd ROT Y ¡Æ¢®¨ùO
DMOV      D004424 D002274	// R_2nd ROT Y ¡Æ¡§¨ùO
DMOV      D004444 D002262	// R_2nd ROT Y ¢¬nC¡ÍA¡×A¢®
DMOV      D004464 D002264	// R_2nd ROT Y ¢¬nC¡Í¨ùO¥ì¥ì
; L89
LOAD NOT  M00600	// EMERGENCY ALARM
AND NOT   D001260.6	// R_3rd SPK Y SVD BUSY
AND NOT   D001260.A	// R_3rd SPK Y WARNING
AND NOT   D001260.B	// R_3rd SPK Y MODULE ERR
AND NOT   D001260.C	// R_3rd SPK Y SVD ERR
AND NOT   M02141	// T)R_3rd SPK Y JOG-
AND NOT   M02142	// T)R_3rd SPK Y JOG+
AND NOT   M02143	// T)R_3rd SPK Y SERVO ON
AND NOT   M0314C	// R_3rd SPK Y HOME->
AND NOT   M00743	// R_3rd SPK Y NOT MV
NOT
OUT       M0164C	// R_3rd SPK Y HOLD CUT
; L90
LOAD NOT  M03140	// -
AND NOT   M03141	// -
AND NOT   M03142	// -
AND NOT   M03143	// -
AND NOT   M03144	// -
AND NOT   M03145	// -
AND NOT   M0314A	// -
AND NOT   M01645	// R_3rd SPK Y INITIAL ->
NOT
OUTP      M0164D	// R_3rd SPK Y START 1PLS
; L91
LOAD      D001260.7	// R_3rd SPK Y A¡×A¢®¡ÆaA¢´ ¢¯I¡¤a
OUTP      M0164E	// R_3rd SPK Y POS OK PLS
; L92
LOAD      M0164D	// R_3rd SPK Y START 1PLS
LOAD      M0164F	// R_3rd SPK Y MOVE HOLD
AND NOT   M0164E	// R_3rd SPK Y POS OK PLS
AND NOT   M0164C	// R_3rd SPK Y HOLD CUT
OR LOAD
OUT       M0164F	// R_3rd SPK Y MOVE HOLD
OUT       D002260.7	// R_3rd SPK Y ABS POS MV
; L94
LOAD NOT  D002260.E	// R_3rd SPK Y ¨¬n¡íoA¢´Ao
TON       T0764 10	// R_3rd SPK Y ¨¬n¡íoA¢´Ao OFF
; L95
LOAD      M00600	// EMERGENCY ALARM
OR        M0214F	// T)R_3rd SPK Y STOP
LOAD      D001260.6	// R_3rd SPK Y SVD BUSY
AND NOT   P0008A	// R_2nd SUPPORT BW
OR LOAD
AND       T0764	// R_3rd SPK Y ¨¬n¡íoA¢´Ao OFF
OUT       D002260.E	// R_3rd SPK Y ¨¬n¡íoA¢´Ao
; L98
LOAD NOT  D001260.E	// R_3rd SPK Y ¡íoCN¢¬¢ç©öI¨¡¢ç
AND NOT   D001260.F	// R_3rd SPK Y CICN¢¬¢ç©öI¨¡¢ç
TON       T0914 2	// R_3rd SPK Y LMT RST TM

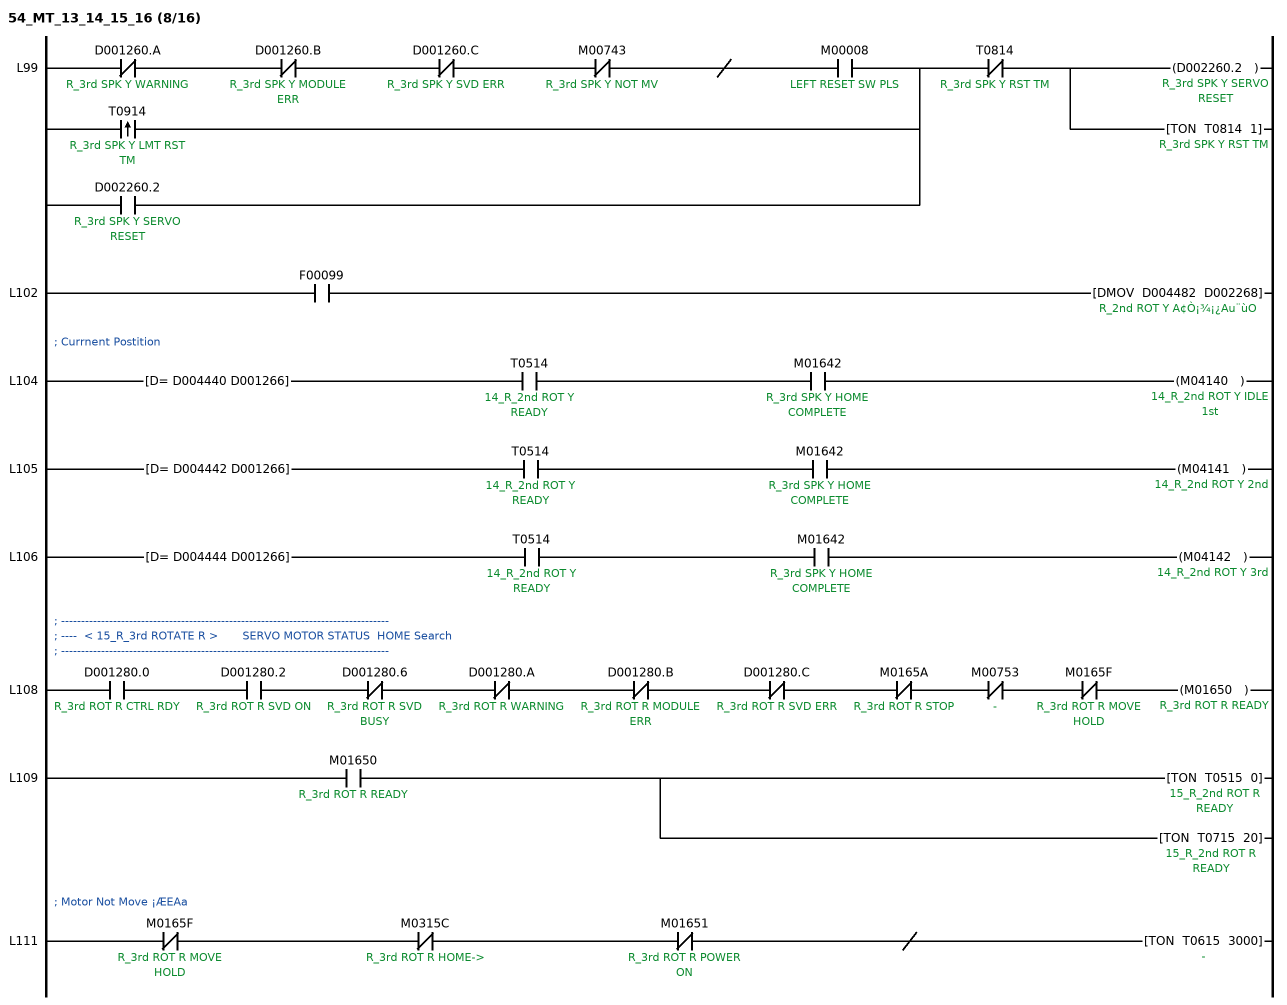
; L99
LOAD NOT  D001260.A	// R_3rd SPK Y WARNING
AND NOT   D001260.B	// R_3rd SPK Y MODULE ERR
AND NOT   D001260.C	// R_3rd SPK Y SVD ERR
AND NOT   M00743	// R_3rd SPK Y NOT MV
NOT
AND       M00008	// LEFT RESET SW PLS
ORP       T0914	// R_3rd SPK Y LMT RST TM
OR        D002260.2	// R_3rd SPK Y SERVO RESET
AND NOT   T0814	// R_3rd SPK Y RST TM
OUT       D002260.2	// R_3rd SPK Y SERVO RESET
TON       T0814 1	// R_3rd SPK Y RST TM
; L102
LOAD      F00099
DMOV      D004482 D002268	// R_2nd ROT Y A¢Ò¡¾¡¿Au¨ùO
// Currnent Postition
; L104
LOADD=    D004440 D001266
AND       T0514	// 14_R_2nd ROT Y READY
AND       M01642	// R_3rd SPK Y HOME COMPLETE
OUT       M04140	// 14_R_2nd ROT Y IDLE 1st
; L105
LOADD=    D004442 D001266
AND       T0514	// 14_R_2nd ROT Y READY
AND       M01642	// R_3rd SPK Y HOME COMPLETE
OUT       M04141	// 14_R_2nd ROT Y 2nd
; L106
LOADD=    D004444 D001266
AND       T0514	// 14_R_2nd ROT Y READY
AND       M01642	// R_3rd SPK Y HOME COMPLETE
OUT       M04142	// 14_R_2nd ROT Y 3rd
// ----------------------------------------------------------------------------------
// 
// ----  < 15_R_3rd ROTATE R >       SERVO MOTOR STATUS  HOME Search
// 
// ----------------------------------------------------------------------------------
; L108
LOAD      D001280.0	// R_3rd ROT R CTRL RDY
AND       D001280.2	// R_3rd ROT R SVD ON
AND NOT   D001280.6	// R_3rd ROT R SVD BUSY
AND NOT   D001280.A	// R_3rd ROT R WARNING
AND NOT   D001280.B	// R_3rd ROT R MODULE ERR
AND NOT   D001280.C	// R_3rd ROT R SVD ERR
AND NOT   M0165A	// R_3rd ROT R STOP
AND NOT   M00753	// -
AND NOT   M0165F	// R_3rd ROT R MOVE HOLD
OUT       M01650	// R_3rd ROT R READY
; L109
LOAD      M01650	// R_3rd ROT R READY
TON       T0515 0	// 15_R_2nd ROT R READY
TON       T0715 20	// 15_R_2nd ROT R READY
; L111
LOAD NOT  M0165F	// R_3rd ROT R MOVE HOLD
AND NOT   M0315C	// R_3rd ROT R HOME->
AND NOT   M01651	// R_3rd ROT R POWER ON
NOT
TON       T0615 3000	// -
// output comment: Motor Not Move ¡ÆEAa

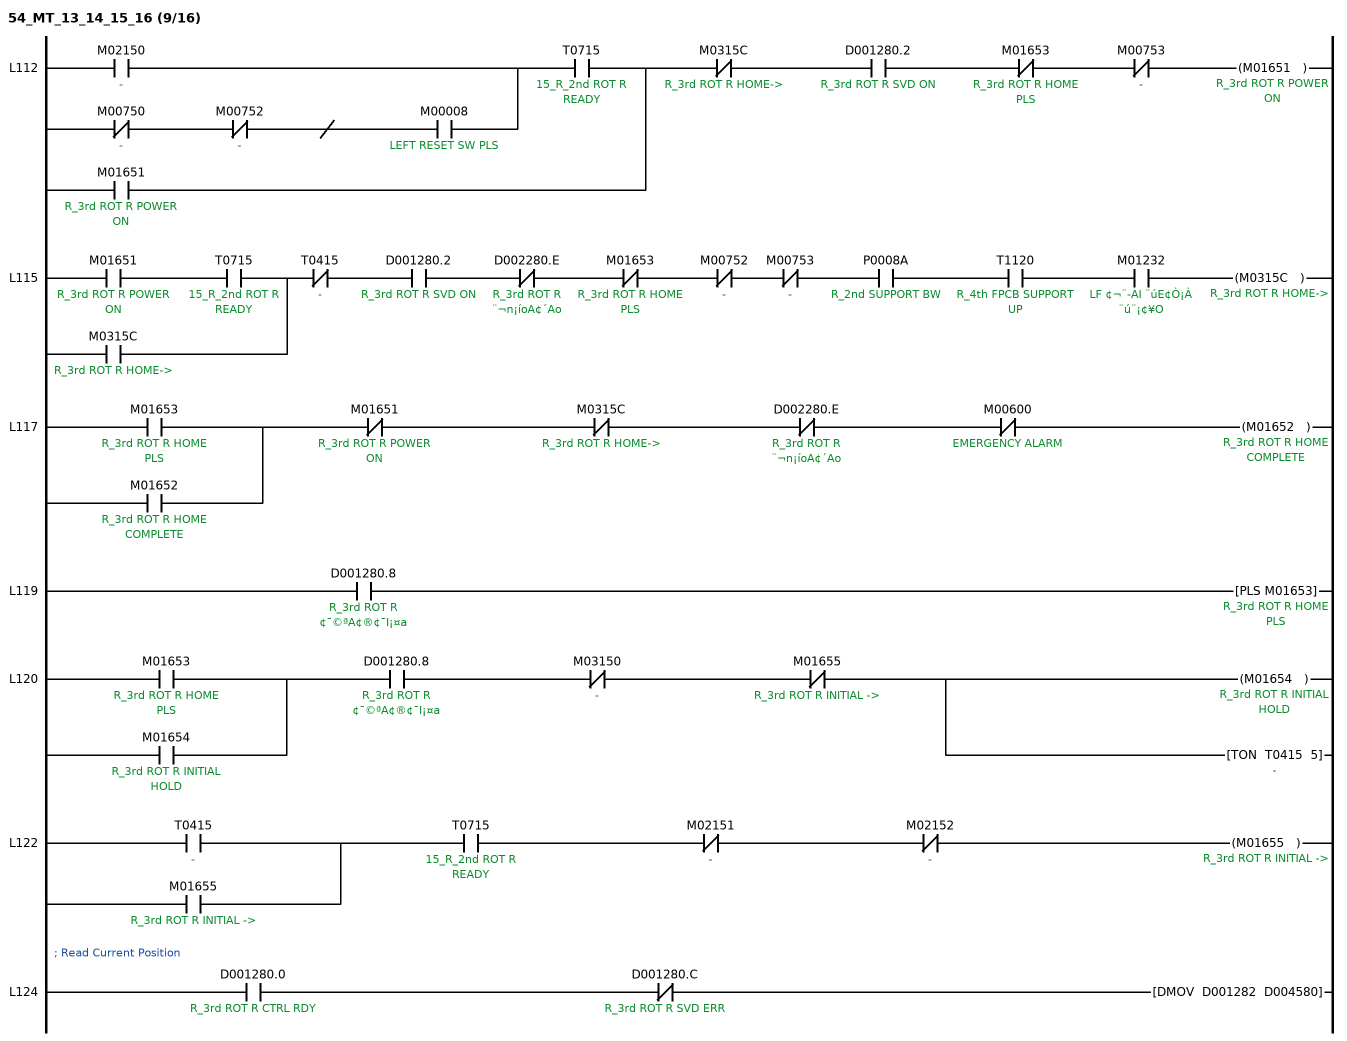
; L112
LOAD      M02150	// -
LOAD NOT  M00750	// -
AND NOT   M00752	// -
NOT
AND       M00008	// LEFT RESET SW PLS
OR LOAD
AND       T0715	// 15_R_2nd ROT R READY
OR        M01651	// R_3rd ROT R POWER ON
AND NOT   M0315C	// R_3rd ROT R HOME->
AND       D001280.2	// R_3rd ROT R SVD ON
AND NOT   M01653	// R_3rd ROT R HOME PLS
AND NOT   M00753	// -
OUT       M01651	// R_3rd ROT R POWER ON
; L115
LOAD      M01651	// R_3rd ROT R POWER ON
AND       T0715	// 15_R_2nd ROT R READY
OR        M0315C	// R_3rd ROT R HOME->
AND NOT   T0415	// -
AND       D001280.2	// R_3rd ROT R SVD ON
AND NOT   D002280.E	// R_3rd ROT R ¨¬n¡íoA¢´Ao
AND NOT   M01653	// R_3rd ROT R HOME PLS
AND NOT   M00752	// -
AND NOT   M00753	// -
AND       P0008A	// R_2nd SUPPORT BW
AND       T1120	// R_4th FPCB SUPPORT UP
AND       M01232	// LF ¢¬¨­AI ¨úE¢Ò¡À ¨ú¨¡¢¥O
OUT       M0315C	// R_3rd ROT R HOME->
; L117
LOAD      M01653	// R_3rd ROT R HOME PLS
OR        M01652	// R_3rd ROT R HOME COMPLETE
AND NOT   M01651	// R_3rd ROT R POWER ON
AND NOT   M0315C	// R_3rd ROT R HOME->
AND NOT   D002280.E	// R_3rd ROT R ¨¬n¡íoA¢´Ao
AND NOT   M00600	// EMERGENCY ALARM
OUT       M01652	// R_3rd ROT R HOME COMPLETE
; L119
LOAD      D001280.8	// R_3rd ROT R ¢¯©ªA¢®¢¯I¡¤a
OUTP      M01653	// R_3rd ROT R HOME PLS
; L120
LOAD      M01653	// R_3rd ROT R HOME PLS
OR        M01654	// R_3rd ROT R INITIAL HOLD
AND       D001280.8	// R_3rd ROT R ¢¯©ªA¢®¢¯I¡¤a
AND NOT   M03150	// -
AND NOT   M01655	// R_3rd ROT R INITIAL ->
OUT       M01654	// R_3rd ROT R INITIAL HOLD
TON       T0415 5	// -
; L122
LOAD      T0415	// -
OR        M01655	// R_3rd ROT R INITIAL ->
AND       T0715	// 15_R_2nd ROT R READY
AND NOT   M02151	// -
AND NOT   M02152	// -
OUT       M01655	// R_3rd ROT R INITIAL ->
; L124
LOAD      D001280.0	// R_3rd ROT R CTRL RDY
AND NOT   D001280.C	// R_3rd ROT R SVD ERR
DMOV      D001282 D004580
// output comment: Read Current Position

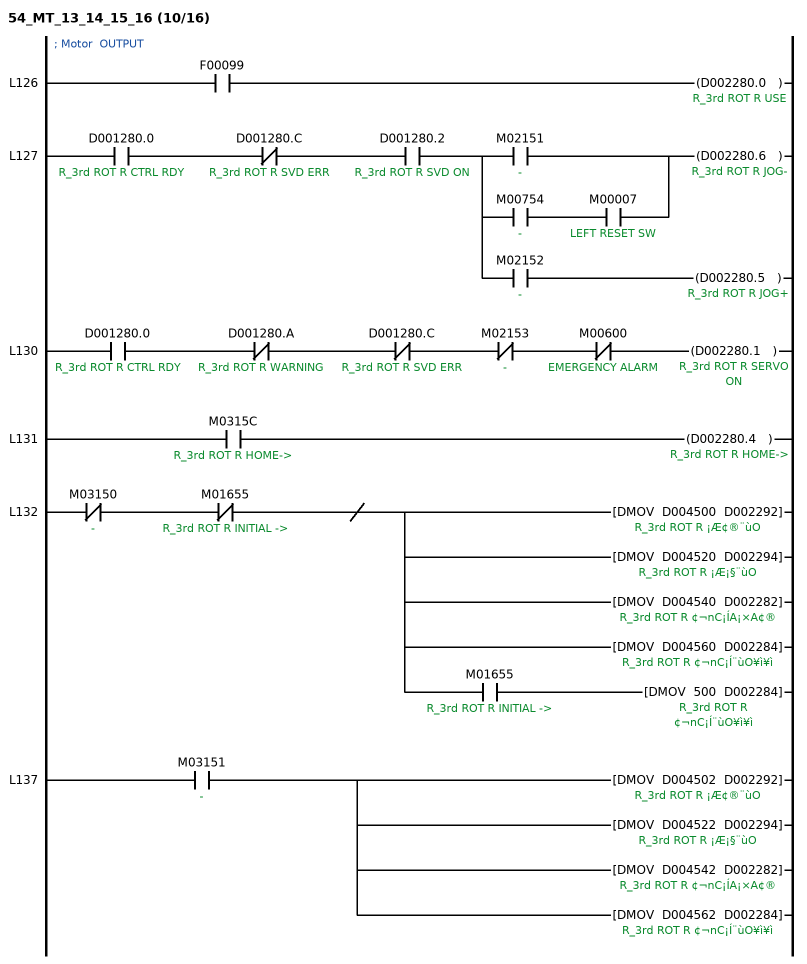
//  Motor  OUTPUT
; L126
LOAD      F00099
OUT       D002280.0	// R_3rd ROT R USE
; L127
LOAD      D001280.0	// R_3rd ROT R CTRL RDY
AND NOT   D001280.C	// R_3rd ROT R SVD ERR
AND       D001280.2	// R_3rd ROT R SVD ON
MPUSH
LOAD      M02151	// -
LOAD      M00754	// -
AND       M00007	// LEFT RESET SW
OR LOAD
AND LOAD
OUT       D002280.6	// R_3rd ROT R JOG-
MPOP
AND       M02152	// -
OUT       D002280.5	// R_3rd ROT R JOG+
; L130
LOAD      D001280.0	// R_3rd ROT R CTRL RDY
AND NOT   D001280.A	// R_3rd ROT R WARNING
AND NOT   D001280.C	// R_3rd ROT R SVD ERR
AND NOT   M02153	// -
AND NOT   M00600	// EMERGENCY ALARM
OUT       D002280.1	// R_3rd ROT R SERVO ON
; L131
LOAD      M0315C	// R_3rd ROT R HOME->
OUT       D002280.4	// R_3rd ROT R HOME->
; L132
LOAD NOT  M03150	// -
AND NOT   M01655	// R_3rd ROT R INITIAL ->
NOT
DMOV      D004500 D002292	// R_3rd ROT R ¡Æ¢®¨ùO
DMOV      D004520 D002294	// R_3rd ROT R ¡Æ¡§¨ùO
DMOV      D004540 D002282	// R_3rd ROT R ¢¬nC¡ÍA¡×A¢®
DMOV      D004560 D002284	// R_3rd ROT R ¢¬nC¡Í¨ùO¥ì¥ì
AND       M01655	// R_3rd ROT R INITIAL ->
DMOV      500 D002284	// R_3rd ROT R ¢¬nC¡Í¨ùO¥ì¥ì
; L137
LOAD      M03151	// -
DMOV      D004502 D002292	// R_3rd ROT R ¡Æ¢®¨ùO
DMOV      D004522 D002294	// R_3rd ROT R ¡Æ¡§¨ùO
DMOV      D004542 D002282	// R_3rd ROT R ¢¬nC¡ÍA¡×A¢®
DMOV      D004562 D002284	// R_3rd ROT R ¢¬nC¡Í¨ùO¥ì¥ì

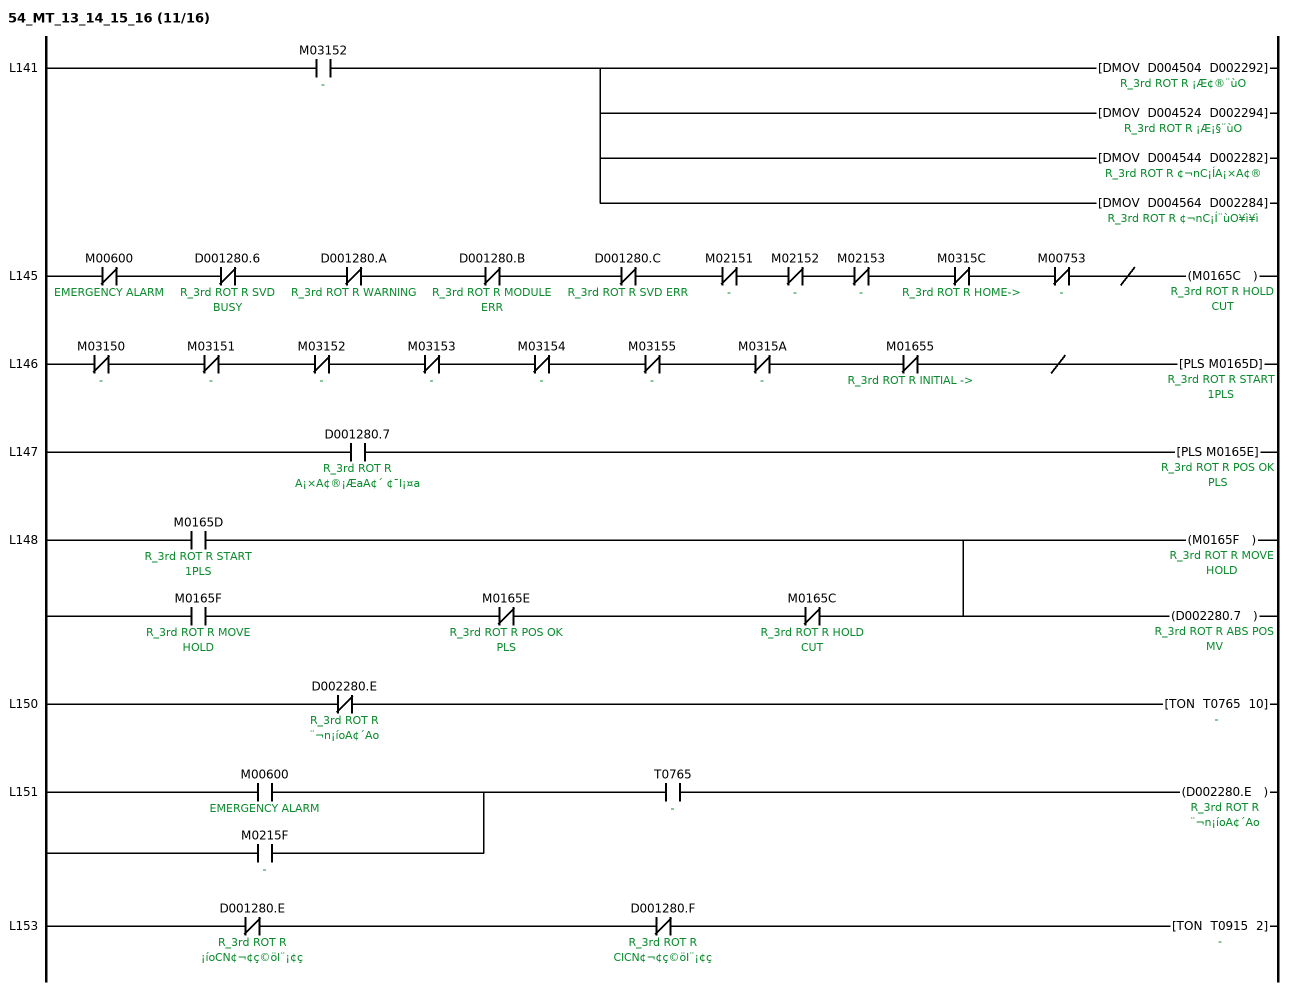
; L141
LOAD      M03152	// -
DMOV      D004504 D002292	// R_3rd ROT R ¡Æ¢®¨ùO
DMOV      D004524 D002294	// R_3rd ROT R ¡Æ¡§¨ùO
DMOV      D004544 D002282	// R_3rd ROT R ¢¬nC¡ÍA¡×A¢®
DMOV      D004564 D002284	// R_3rd ROT R ¢¬nC¡Í¨ùO¥ì¥ì
; L145
LOAD NOT  M00600	// EMERGENCY ALARM
AND NOT   D001280.6	// R_3rd ROT R SVD BUSY
AND NOT   D001280.A	// R_3rd ROT R WARNING
AND NOT   D001280.B	// R_3rd ROT R MODULE ERR
AND NOT   D001280.C	// R_3rd ROT R SVD ERR
AND NOT   M02151	// -
AND NOT   M02152	// -
AND NOT   M02153	// -
AND NOT   M0315C	// R_3rd ROT R HOME->
AND NOT   M00753	// -
NOT
OUT       M0165C	// R_3rd ROT R HOLD CUT
; L146
LOAD NOT  M03150	// -
AND NOT   M03151	// -
AND NOT   M03152	// -
AND NOT   M03153	// -
AND NOT   M03154	// -
AND NOT   M03155	// -
AND NOT   M0315A	// -
AND NOT   M01655	// R_3rd ROT R INITIAL ->
NOT
OUTP      M0165D	// R_3rd ROT R START 1PLS
; L147
LOAD      D001280.7	// R_3rd ROT R A¡×A¢®¡ÆaA¢´ ¢¯I¡¤a
OUTP      M0165E	// R_3rd ROT R POS OK PLS
; L148
LOAD      M0165D	// R_3rd ROT R START 1PLS
LOAD      M0165F	// R_3rd ROT R MOVE HOLD
AND NOT   M0165E	// R_3rd ROT R POS OK PLS
AND NOT   M0165C	// R_3rd ROT R HOLD CUT
OR LOAD
OUT       M0165F	// R_3rd ROT R MOVE HOLD
OUT       D002280.7	// R_3rd ROT R ABS POS MV
; L150
LOAD NOT  D002280.E	// R_3rd ROT R ¨¬n¡íoA¢´Ao
TON       T0765 10	// -
; L151
LOAD      M00600	// EMERGENCY ALARM
OR        M0215F	// -
AND       T0765	// -
OUT       D002280.E	// R_3rd ROT R ¨¬n¡íoA¢´Ao
; L153
LOAD NOT  D001280.E	// R_3rd ROT R ¡íoCN¢¬¢ç©öI¨¡¢ç
AND NOT   D001280.F	// R_3rd ROT R CICN¢¬¢ç©öI¨¡¢ç
TON       T0915 2	// -

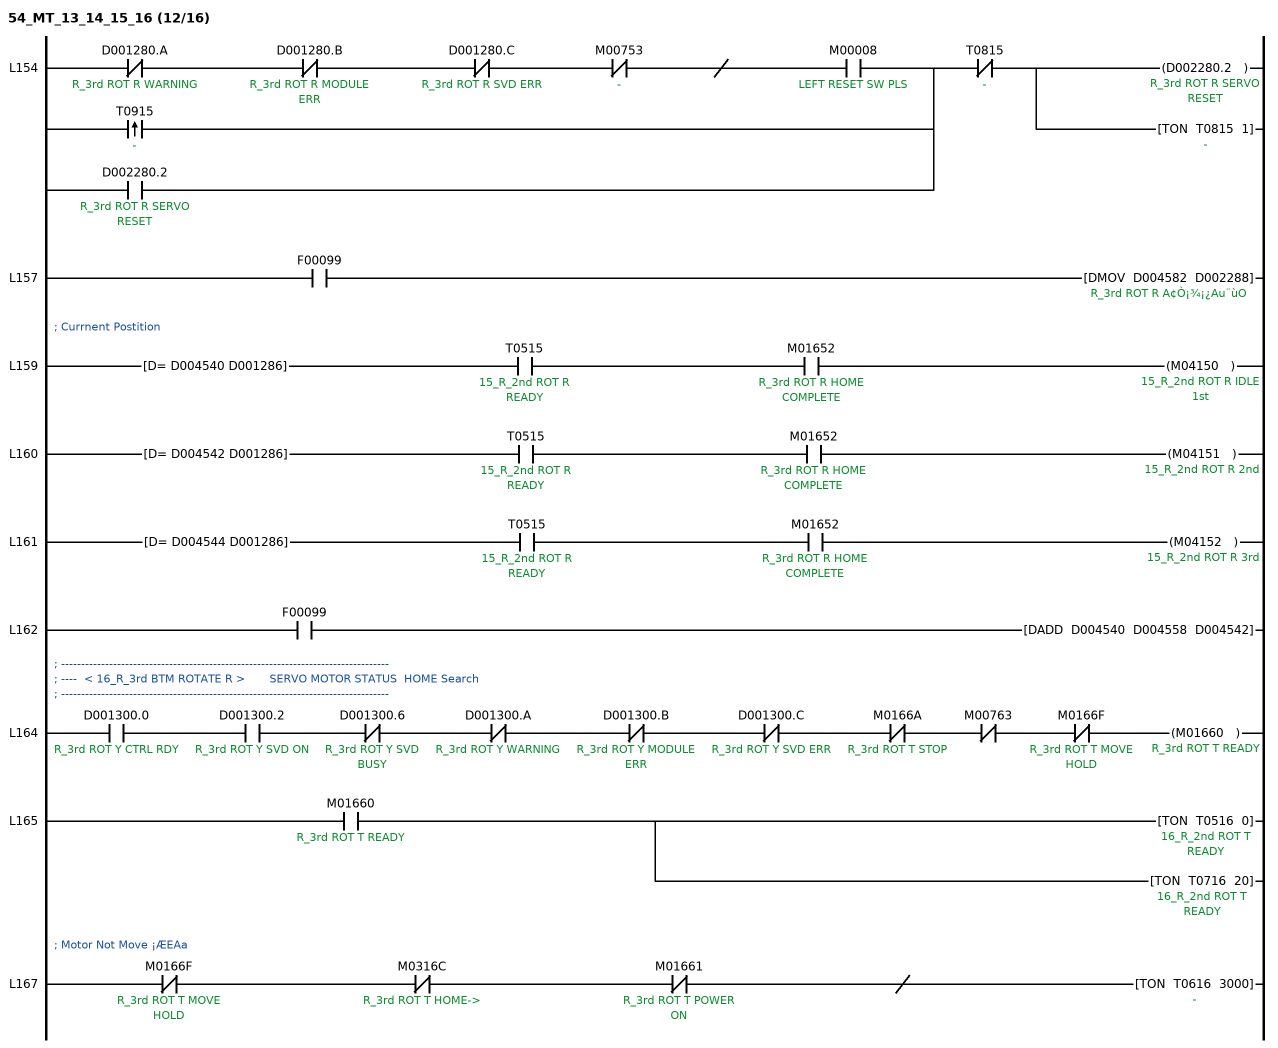
; L154
LOAD NOT  D001280.A	// R_3rd ROT R WARNING
AND NOT   D001280.B	// R_3rd ROT R MODULE ERR
AND NOT   D001280.C	// R_3rd ROT R SVD ERR
AND NOT   M00753	// -
NOT
AND       M00008	// LEFT RESET SW PLS
ORP       T0915	// -
OR        D002280.2	// R_3rd ROT R SERVO RESET
AND NOT   T0815	// -
OUT       D002280.2	// R_3rd ROT R SERVO RESET
TON       T0815 1	// -
; L157
LOAD      F00099
DMOV      D004582 D002288	// R_3rd ROT R A¢Ò¡¾¡¿Au¨ùO
// Currnent Postition
; L159
LOADD=    D004540 D001286
AND       T0515	// 15_R_2nd ROT R READY
AND       M01652	// R_3rd ROT R HOME COMPLETE
OUT       M04150	// 15_R_2nd ROT R IDLE 1st
; L160
LOADD=    D004542 D001286
AND       T0515	// 15_R_2nd ROT R READY
AND       M01652	// R_3rd ROT R HOME COMPLETE
OUT       M04151	// 15_R_2nd ROT R 2nd
; L161
LOADD=    D004544 D001286
AND       T0515	// 15_R_2nd ROT R READY
AND       M01652	// R_3rd ROT R HOME COMPLETE
OUT       M04152	// 15_R_2nd ROT R 3rd
; L162
LOAD      F00099
DADD      D004540 D004558 D004542
// ----------------------------------------------------------------------------------
// 
// ----  < 16_R_3rd BTM ROTATE R >       SERVO MOTOR STATUS  HOME Search
// 
// ----------------------------------------------------------------------------------
; L164
LOAD      D001300.0	// R_3rd ROT Y CTRL RDY
AND       D001300.2	// R_3rd ROT Y SVD ON
AND NOT   D001300.6	// R_3rd ROT Y SVD BUSY
AND NOT   D001300.A	// R_3rd ROT Y WARNING
AND NOT   D001300.B	// R_3rd ROT Y MODULE ERR
AND NOT   D001300.C	// R_3rd ROT Y SVD ERR
AND NOT   M0166A	// R_3rd ROT T STOP
AND NOT   M00763
AND NOT   M0166F	// R_3rd ROT T MOVE HOLD
OUT       M01660	// R_3rd ROT T READY
; L165
LOAD      M01660	// R_3rd ROT T READY
TON       T0516 0	// 16_R_2nd ROT T READY
TON       T0716 20	// 16_R_2nd ROT T READY
; L167
LOAD NOT  M0166F	// R_3rd ROT T MOVE HOLD
AND NOT   M0316C	// R_3rd ROT T HOME->
AND NOT   M01661	// R_3rd ROT T POWER ON
NOT
TON       T0616 3000	// -
// output comment: Motor Not Move ¡ÆEAa

